  MoveC 4849 to (-301.47, 196.97, -44.5) mm, rotated rx -180 ry 0 rz 0.01 deg; joints [33.555, -39.251, 93.109, -140.852, 61.141, 159.518] to (-302.58, 195.21, -44.5) mm, rotated rx -180 ry 0 rz 0.01 deg; joints [33.481, -39.252, 93.114, -140.932, 61.116, 159.56]
  MoveL 4850 to (-302.58, 149.34, -44.5) mm, rotated rx -180 ry 0 rz 0.01 deg; joints [32.097, -40.399, 95.628, -142.863, 61.697, 161.24]
  MoveC 4851 to (-301.48, 145.02, -44.5) mm, rotated rx 180 ry 0 rz 0.01 deg; joints [31.985, -40.546, 95.95, -143.039, 61.798, 161.417] to (-298.46, 141.74, -44.5) mm, rotated rx 180 ry 0 rz 0.01 deg; joints [31.942, -40.745, 96.378, -143.159, 61.967, 161.595]
  MoveC 4852 to (-293.36, 138.32, -44.5) mm, rotated rx -180 ry 0 rz 0.01 deg; joints [31.935, -41.027, 96.986, -143.27, 62.225, 161.82] to (-288.34, 134.8, -44.5) mm, rotated rx 180 ry 0 rz 0.01 deg; joints [31.923, -41.306, 97.589, -143.384, 62.481, 162.044]
  MoveC 4853 to (-283.47, 131.07, -44.5) mm, rotated rx -180 ry 0 rz 0.01 deg; joints [31.901, -41.583, 98.188, -143.506, 62.732, 162.271] to (-278.83, 127.06, -44.5) mm, rotated rx -180 ry 0 rz 0.01 deg; joints [31.866, -41.856, 98.779, -143.64, 62.977, 162.5]
  MoveC 4854 to (-271.87, 120.15, -44.5) mm, rotated rx 180 ry 0 rz 0.01 deg; joints [31.785, -42.282, 99.704, -143.876, 63.353, 162.871] to (-265.5, 112.7, -44.5) mm, rotated rx -180 ry 0 rz 0.01 deg; joints [31.673, -42.694, 100.6, -144.136, 63.71, 163.243]
  MoveC 4855 to (-259.72, 104.78, -44.5) mm, rotated rx -180 ry 0 rz 0.01 deg; joints [31.534, -43.089, 101.465, -144.418, 64.048, 163.615] to (-254.52, 96.46, -44.5) mm, rotated rx 180 ry 0 rz 0.01 deg; joints [31.369, -43.468, 102.295, -144.719, 64.366, 163.983]
  MoveL 4856 to (-242.31, 74.19, -44.5) mm, rotated rx 180 ry 0 rz 0.01 deg; joints [30.883, -44.399, 104.348, -145.536, 65.145, 164.917]
  MoveC 4857 to (-239.21, 71.08, -44.5) mm, rotated rx 180 ry 0 rz 0.01 deg; joints [30.842, -44.578, 104.742, -145.635, 65.311, 165.069] to (-234.96, 69.94, -44.5) mm, rotated rx 180 ry 0 rz 0.01 deg; joints [30.888, -44.757, 105.133, -145.641, 65.498, 165.18]
  MoveL 4858 to (-158.58, 69.94, -44.5) mm, rotated rx 180 ry 0 rz 0.01 deg; joints [32.47, -47.442, 110.991, -144.753, 68.529, 166.484]
  MoveC 4859 to (-154.33, 71.08, -44.5) mm, rotated rx -180 ry 0 rz 0.01 deg; joints [32.601, -47.562, 111.253, -144.649, 68.678, 166.521] to (-151.22, 74.19, -44.5) mm, rotated rx -180 ry 0 rz 0.01 deg; joints [32.775, -47.603, 111.336, -144.479, 68.757, 166.48]
  MoveL 4860 to (-138.74, 96.86, -44.5) mm, rotated rx 180 ry 0 rz 0.01 deg; joints [33.818, -47.543, 111.16, -143.372, 68.936, 166.005]
  MoveC 4861 to (-132.58, 106.47, -44.5) mm, rotated rx -180 ry 0 rz 0.01 deg; joints [34.279, -47.541, 111.137, -142.891, 69.042, 165.816] to (-125.56, 115.48, -44.5) mm, rotated rx 180 ry 0 rz 0.01 deg; joints [34.74, -47.577, 111.197, -142.423, 69.186, 165.658]
  MoveC 4862 to (-117.83, 123.88, -44.5) mm, rotated rx -180 ry 0 rz 0.01 deg; joints [35.197, -47.646, 111.333, -141.967, 69.362, 165.53] to (-109.5, 131.68, -44.5) mm, rotated rx 180 ry 0 rz 0.01 deg; joints [35.65, -47.744, 111.532, -141.526, 69.566, 165.429]
  MoveC 4863 to (-106.07, 134.44, -44.5) mm, rotated rx 180 ry 0 rz 0.01 deg; joints [35.822, -47.793, 111.635, -141.362, 69.656, 165.402] to (-102.44, 136.93, -44.5) mm, rotated rx -180 ry 0 rz 0.01 deg; joints [35.99, -47.854, 111.765, -141.206, 69.756, 165.386]
  MoveC 4864 to (-98.74, 139.29, -44.5) mm, rotated rx 180 ry 0 rz 0.01 deg; joints [36.157, -47.92, 111.906, -141.053, 69.86, 165.375] to (-95.05, 141.69, -44.5) mm, rotated rx 180 ry 0 rz 0.01 deg; joints [36.324, -47.984, 112.042, -140.898, 69.962, 165.363]
  MoveC 4865 to (-92.03, 145, -44.5) mm, rotated rx -180 ry 0 rz 0.01 deg; joints [36.505, -48.006, 112.083, -140.717, 70.027, 165.311] to (-90.94, 149.34, -44.5) mm, rotated rx 180 ry 0 rz 0.01 deg; joints [36.673, -47.942, 111.934, -140.525, 70.008, 165.193]
  MoveL 4866 to (-90.94, 195.21, -44.5) mm, rotated rx 180 ry 0 rz 0.01 deg; joints [38.14, -46.86, 109.476, -138.699, 69.387, 163.706]
  MoveC 4867 to (-92.04, 196.97, -44.5) mm, rotated rx 180 ry 0 rz 0.01 deg; joints [38.168, -46.782, 109.301, -138.647, 69.323, 163.628] to (-94.11, 196.74, -44.5) mm, rotated rx -180 ry 0 rz 0.01 deg; joints [38.11, -46.721, 109.169, -138.688, 69.251, 163.599]
  MoveC 4868 to (-101.15, 191.39, -44.5) mm, rotated rx 180 ry 0 rz 0.01 deg; joints [37.77, -46.624, 108.966, -139.008, 69.068, 163.652] to (-108.38, 186.3, -44.5) mm, rotated rx 180 ry 0 rz 0.01 deg; joints [37.435, -46.512, 108.731, -139.319, 68.873, 163.692]
  MoveC 4869 to (-115.9, 181.63, -44.5) mm, rotated rx -180 ry 0 rz 0.01 deg; joints [37.108, -46.378, 108.447, -139.615, 68.66, 163.712] to (-123.75, 177.56, -44.5) mm, rotated rx 180 ry 0 rz 0.01 deg; joints [36.793, -46.216, 108.102, -139.891, 68.424, 163.706]
  MoveC 4870 to (-133.69, 173.48, -44.5) mm, rotated rx 180 ry 0 rz 0.01 deg; joints [36.431, -45.983, 107.602, -140.194, 68.109, 163.663] to (-143.98, 170.42, -44.5) mm, rotated rx -180 ry 0 rz 0.01 deg; joints [36.095, -45.71, 107.013, -140.457, 67.764, 163.578]
  MoveC 4871 to (-154.47, 168.17, -44.5) mm, rotated rx -180 ry 0 rz 0.01 deg; joints [35.784, -45.408, 106.36, -140.686, 67.398, 163.463] to (-165.06, 166.49, -44.5) mm, rotated rx -180 ry 0 rz 0.01 deg; joints [35.491, -45.084, 105.661, -140.888, 67.016, 163.325]
  MoveC 4872 to (-171.83, 165.83, -44.5) mm, rotated rx 180 ry 0 rz 0.01 deg; joints [35.319, -44.866, 105.189, -140.998, 66.766, 163.223] to (-178.62, 165.62, -44.5) mm, rotated rx 180 ry 0 rz 0.01 deg; joints [35.161, -44.635, 104.688, -141.088, 66.507, 163.106]
  MoveL 4873 to (-214.9, 165.62, -44.5) mm, rotated rx 180 ry 0 rz 0.01 deg; joints [34.374, -43.342, 101.899, -141.486, 65.088, 162.423]
  MoveC 4874 to (-230.33, 166.55, -44.5) mm, rotated rx 180 ry 0 rz 0.01 deg; joints [34.077, -42.755, 100.635, -141.597, 64.461, 162.093] to (-245.53, 169.34, -44.5) mm, rotated rx 180 ry 0 rz 0.01 deg; joints [33.847, -42.121, 99.271, -141.618, 63.812, 161.697]
  MoveL 4875 to (-245.78, 169.4, -44.5) mm, rotated rx 180 ry 0 rz 0.01 deg; joints [33.844, -42.11, 99.247, -141.618, 63.801, 161.69]
  MoveC 4876 to (-248.84, 171.23, -44.5) mm, rotated rx 180 ry 0 rz 0.01 deg; joints [33.837, -41.95, 98.902, -141.568, 63.653, 161.564] to (-250.35, 174.46, -44.5) mm, rotated rx 180 ry 0 rz 0.01 deg; joints [33.905, -41.814, 98.605, -141.447, 63.55, 161.42]
  MoveC 4877 to (-251.79, 177.71, -44.5) mm, rotated rx 180 ry 0 rz 0.01 deg; joints [33.974, -41.68, 98.312, -141.325, 63.45, 161.277] to (-254.71, 179.71, -44.5) mm, rotated rx 180 ry 0 rz 0.01 deg; joints [33.976, -41.519, 97.966, -141.265, 63.306, 161.146]
  MoveC 4878 to (-260.13, 181.68, -44.5) mm, rotated rx -180 ry 0 rz 0.01 deg; joints [33.925, -41.263, 97.416, -141.226, 63.059, 160.964] to (-265.46, 183.91, -44.5) mm, rotated rx 180 ry 0 rz 0.01 deg; joints [33.883, -41.003, 96.857, -141.174, 62.811, 160.774]
  MoveC 4879 to (-287.95, 196.94, -44.5) mm, rotated rx -180 ry 0 rz 0.01 deg; joints [33.822, -39.793, 94.259, -140.779, 61.711, 159.818] to (-307.16, 214.45, -44.5) mm, rotated rx -180 ry 0 rz 0.01 deg; joints [33.958, -38.561, 91.618, -140.142, 60.675, 158.723]
  MoveC 4880 to (-309.04, 214.92, -44.5) mm, rotated rx -180 ry 0 rz 0.01 deg; joints [33.934, -38.472, 91.428, -140.13, 60.589, 158.662] to (-310.14, 213.32, -44.5) mm, rotated rx 180 ry 0 rz 0.01 deg; joints [33.866, -38.469, 91.425, -140.203, 60.563, 158.698]
  MoveL 4881 to (-310.14, 144.76, -44.5) mm, rotated rx 180 ry 0 rz 0.01 deg; joints [31.812, -40.207, 95.227, -143.1, 61.432, 161.245]
  MoveC 4882 to (-309.04, 140.62, -44.5) mm, rotated rx 180 ry 0 rz 0.01 deg; joints [31.706, -40.35, 95.539, -143.268, 61.531, 161.416] to (-306.04, 137.56, -44.5) mm, rotated rx -180 ry 0 rz 0.01 deg; joints [31.668, -40.543, 95.955, -143.38, 61.697, 161.586]
  MoveC 4883 to (-295.24, 130.34, -44.5) mm, rotated rx 180 ry 0 rz 0.01 deg; joints [31.651, -41.141, 97.243, -143.617, 62.246, 162.06] to (-285.24, 122.05, -44.5) mm, rotated rx 180 ry 0 rz 0.01 deg; joints [31.585, -41.724, 98.504, -143.896, 62.771, 162.545]
  MoveC 4884 to (-276.09, 112.83, -44.5) mm, rotated rx 180 ry 0 rz 0.01 deg; joints [31.471, -42.287, 99.727, -144.215, 63.269, 163.036] to (-267.8, 102.84, -44.5) mm, rotated rx 180 ry 0 rz 0.01 deg; joints [31.314, -42.827, 100.905, -144.567, 63.738, 163.527]
  MoveC 4885 to (-264.28, 97.87, -44.5) mm, rotated rx -180 ry 0 rz 0.01 deg; joints [31.223, -43.07, 101.436, -144.745, 63.946, 163.757] to (-261.08, 92.69, -44.5) mm, rotated rx -180 ry 0 rz 0.01 deg; joints [31.119, -43.304, 101.95, -144.934, 64.143, 163.985]
  MoveL 4886 to (-246.68, 66.63, -44.5) mm, rotated rx 180 ry 0 rz 0.01 deg; joints [30.548, -44.397, 104.357, -145.893, 65.06, 165.077]
  MoveC 4887 to (-243.58, 63.52, -44.5) mm, rotated rx -180 ry 0 rz 0.01 deg; joints [30.506, -44.576, 104.751, -145.993, 65.226, 165.229] to (-239.33, 62.38, -44.5) mm, rotated rx -180 ry 0 rz 0.01 deg; joints [30.551, -44.755, 105.142, -146, 65.414, 165.338]
  MoveL 4888 to (-154.21, 62.38, -44.5) mm, rotated rx -180 ry 0 rz 0.01 deg; joints [32.307, -47.744, 111.671, -145.008, 68.796, 166.781]
  MoveC 4889 to (-149.96, 63.52, -44.5) mm, rotated rx -180 ry 0 rz 0.01 deg; joints [32.438, -47.864, 111.932, -144.903, 68.945, 166.817] to (-146.85, 66.63, -44.5) mm, rotated rx -180 ry 0 rz 0.01 deg; joints [32.613, -47.904, 112.016, -144.732, 69.024, 166.777]
  MoveL 4890 to (-132.19, 93.08, -44.5) mm, rotated rx 180 ry 0 rz 0.01 deg; joints [33.839, -47.841, 111.823, -143.435, 69.234, 166.23]
  MoveC 4891 to (-123.29, 106.29, -44.5) mm, rotated rx 180 ry 0 rz 0.01 deg; joints [34.486, -47.852, 111.819, -142.764, 69.393, 165.979] to (-112.66, 118.15, -44.5) mm, rotated rx 180 ry 0 rz 0.01 deg; joints [35.128, -47.941, 111.992, -142.122, 69.631, 165.795]
  MoveC 4892 to (-100.62, 128.57, -44.5) mm, rotated rx -180 ry 0 rz 0.01 deg; joints [35.758, -48.1, 112.322, -141.515, 69.936, 165.678] to (-87.47, 137.53, -44.5) mm, rotated rx -180 ry 0 rz 0.01 deg; joints [36.371, -48.319, 112.79, -140.944, 70.295, 165.623]
  MoveC 4893 to (-84.47, 140.62, -44.5) mm, rotated rx 180 ry 0 rz 0.01 deg; joints [36.545, -48.345, 112.841, -140.772, 70.362, 165.578] to (-83.38, 144.77, -44.5) mm, rotated rx 180 ry 0 rz 0.01 deg; joints [36.708, -48.286, 112.701, -140.587, 70.345, 165.466]
  MoveL 4894 to (-83.38, 213.32, -44.5) mm, rotated rx 180 ry 0 rz 0.01 deg; joints [38.891, -46.656, 108.998, -137.867, 69.413, 163.235]
  MoveC 4895 to (-84.48, 214.91, -44.5) mm, rotated rx -180 ry 0 rz 0.01 deg; joints [38.913, -46.582, 108.832, -137.822, 69.352, 163.161] to (-86.36, 214.45, -44.5) mm, rotated rx 180 ry 0 rz 0.01 deg; joints [38.852, -46.533, 108.727, -137.87, 69.291, 163.143]
  MoveC 4896 to (-103.09, 198.94, -44.5) mm, rotated rx 180 ry 0 rz 0.01 deg; joints [37.959, -46.377, 108.414, -138.738, 68.896, 163.365] to (-122.53, 187, -44.5) mm, rotated rx -180 ry 0 rz 0.01 deg; joints [37.119, -46.03, 107.679, -139.497, 68.343, 163.415]
  MoveC 4897 to (-143.76, 178.74, -44.5) mm, rotated rx -180 ry 0 rz 0.01 deg; joints [36.363, -45.519, 106.583, -140.12, 67.662, 163.306] to (-166.04, 173.99, -44.5) mm, rotated rx 180 ry 0 rz 0.01 deg; joints [35.705, -44.872, 105.187, -140.597, 66.881, 163.057]
  MoveC 4898 to (-172.31, 173.38, -44.5) mm, rotated rx 180 ry 0 rz 0.01 deg; joints [35.545, -44.669, 104.749, -140.698, 66.648, 162.962] to (-178.62, 173.18, -44.5) mm, rotated rx 180 ry 0 rz 0.01 deg; joints [35.398, -44.454, 104.284, -140.781, 66.409, 162.851]
  MoveL 4899 to (-214.9, 173.18, -44.5) mm, rotated rx 180 ry 0 rz 0.01 deg; joints [34.608, -43.16, 101.494, -141.176, 64.991, 162.164]
  MoveC 4900 to (-235.07, 174.82, -44.5) mm, rotated rx -180 ry 0 rz 0.01 deg; joints [34.233, -42.378, 99.812, -141.301, 64.164, 161.713] to (-254.71, 179.71, -44.5) mm, rotated rx 180 ry 0 rz 0.01 deg; joints [33.976, -41.519, 97.966, -141.265, 63.306, 161.146]
  MoveC 4901 to (-257.49, 181.72, -44.5) mm, rotated rx 180 ry 0 rz 0.01 deg; joints [33.979, -41.363, 97.63, -141.204, 63.166, 161.017] to (-258.67, 184.93, -44.5) mm, rotated rx -180 ry 0 rz 0.01 deg; joints [34.053, -41.238, 97.357, -141.08, 63.077, 160.878]
  MoveC 4902 to (-259.76, 188.16, -44.5) mm, rotated rx -180 ry 0 rz 0.01 deg; joints [34.128, -41.115, 97.089, -140.955, 62.991, 160.739] to (-262.38, 190.33, -44.5) mm, rotated rx -180 ry 0 rz 0.01 deg; joints [34.14, -40.96, 96.754, -140.884, 62.856, 160.606]
  MoveC 4903 to (-291.82, 209.03, -44.5) mm, rotated rx 180 ry 0 rz 0.01 deg; joints [34.103, -39.324, 93.244, -140.294, 61.394, 159.279] to (-314.46, 235.55, -44.5) mm, rotated rx -180 ry 0 rz 0.01 deg; joints [34.426, -37.687, 89.738, -139.276, 60.092, 157.725]
  MoveC 4904 to (-316.16, 236.21, -44.5) mm, rotated rx -180 ry 0 rz 0.01 deg; joints [34.412, -37.599, 89.55, -139.254, 60.011, 157.658] to (-317.25, 234.75, -44.5) mm, rotated rx 180 ry 0 rz 0.01 deg; joints [34.348, -37.593, 89.54, -139.32, 59.982, 157.689]
  MoveL 4905 to (-317.25, 140.22, -44.5) mm, rotated rx -180 ry 0 rz 0.01 deg; joints [31.538, -40.029, 94.857, -143.33, 61.184, 161.257]
  MoveC 4906 to (-316.15, 136.26, -44.5) mm, rotated rx -180 ry 0 rz 0.01 deg; joints [31.437, -40.168, 95.159, -143.491, 61.28, 161.422] to (-313.18, 133.42, -44.5) mm, rotated rx 180 ry 0 rz 0.01 deg; joints [31.406, -40.355, 95.562, -143.595, 61.443, 161.584]
  MoveC 4907 to (-301.85, 126.44, -44.5) mm, rotated rx -180 ry 0 rz 0.01 deg; joints [31.404, -40.971, 96.887, -143.823, 62.014, 162.062] to (-291.44, 118.13, -44.5) mm, rotated rx -180 ry 0 rz 0.01 deg; joints [31.342, -41.572, 98.186, -144.104, 62.558, 162.557]
  MoveC 4908 to (-281.99, 108.76, -44.5) mm, rotated rx 180 ry 0 rz 0.01 deg; joints [31.228, -42.152, 99.444, -144.429, 63.072, 163.059] to (-273.47, 98.55, -44.5) mm, rotated rx 180 ry 0 rz 0.01 deg; joints [31.066, -42.706, 100.653, -144.792, 63.556, 163.562]
  MoveC 4909 to (-270.21, 93.94, -44.5) mm, rotated rx -180 ry 0 rz 0.01 deg; joints [30.982, -42.932, 101.146, -144.958, 63.749, 163.775] to (-267.24, 89.14, -44.5) mm, rotated rx -180 ry 0 rz 0.01 deg; joints [30.884, -43.149, 101.622, -145.134, 63.932, 163.987]
  MoveL 4910 to (-250.77, 59.48, -44.5) mm, rotated rx 180 ry 0 rz 0.01 deg; joints [30.232, -44.394, 104.364, -146.23, 64.981, 165.228]
  MoveC 4911 to (-247.69, 56.39, -44.5) mm, rotated rx 180 ry 0 rz 0.01 deg; joints [30.189, -44.571, 104.754, -146.33, 65.146, 165.378] to (-243.48, 55.27, -44.5) mm, rotated rx 180 ry 0 rz 0.01 deg; joints [30.233, -44.749, 105.143, -146.338, 65.333, 165.486]
  MoveL 4912 to (-150.04, 55.27, -44.5) mm, rotated rx 180 ry 0 rz 0.01 deg; joints [32.152, -48.028, 112.311, -145.247, 69.05, 167.058]
  MoveC 4913 to (-145.85, 56.39, -44.5) mm, rotated rx 180 ry 0 rz 0.01 deg; joints [32.282, -48.145, 112.568, -145.142, 69.197, 167.094] to (-142.78, 59.46, -44.5) mm, rotated rx -180 ry 0 rz 0.01 deg; joints [32.455, -48.186, 112.652, -144.972, 69.275, 167.055]
  MoveL 4914 to (-126.04, 89.52, -44.5) mm, rotated rx 180 ry 0 rz 0.01 deg; joints [33.858, -48.119, 112.443, -143.491, 69.514, 166.441]
  MoveC 4915 to (-117.03, 102.79, -44.5) mm, rotated rx -180 ry 0 rz 0.01 deg; joints [34.513, -48.131, 112.443, -142.814, 69.675, 166.191] to (-106.22, 114.63, -44.5) mm, rotated rx -180 ry 0 rz 0.01 deg; joints [35.162, -48.226, 112.628, -142.167, 69.917, 166.012]
  MoveC 4916 to (-93.89, 124.88, -44.5) mm, rotated rx 180 ry 0 rz 0.01 deg; joints [35.796, -48.397, 112.985, -141.558, 70.233, 165.906] to (-80.33, 133.42, -44.5) mm, rotated rx 180 ry 0 rz 0.01 deg; joints [36.409, -48.637, 113.5, -140.993, 70.61, 165.872]
  MoveC 4917 to (-77.36, 136.28, -44.5) mm, rotated rx 180 ry 0 rz 0.01 deg; joints [36.576, -48.667, 113.56, -140.829, 70.679, 165.834] to (-76.26, 140.26, -44.5) mm, rotated rx -180 ry 0 rz 0.01 deg; joints [36.734, -48.612, 113.431, -140.651, 70.664, 165.728]
  MoveL 4918 to (-76.26, 234.75, -44.5) mm, rotated rx -180 ry 0 rz 0.01 deg; joints [39.726, -46.342, 108.276, -136.917, 69.377, 162.633]
  MoveC 4919 to (-77.36, 236.2, -44.5) mm, rotated rx -180 ry 0 rz 0.01 deg; joints [39.743, -46.27, 108.116, -136.878, 69.318, 162.563] to (-79.06, 235.54, -44.5) mm, rotated rx 180 ry 0 rz 0.01 deg; joints [39.68, -46.233, 108.036, -136.93, 69.267, 162.555]
  MoveC 4920 to (-91.63, 218.9, -44.5) mm, rotated rx -180 ry 0 rz 0.01 deg; joints [38.858, -46.253, 108.107, -137.777, 69.042, 162.897] to (-107.02, 204.82, -44.5) mm, rotated rx 180 ry 0 rz 0.01 deg; joints [38.047, -46.104, 107.809, -138.563, 68.674, 163.097]
  MoveC 4921 to (-124.62, 193.66, -44.5) mm, rotated rx -180 ry 0 rz 0.01 deg; joints [37.278, -45.799, 107.164, -139.261, 68.177, 163.154] to (-143.84, 185.59, -44.5) mm, rotated rx 180 ry 0 rz 0.01 deg; joints [36.575, -45.351, 106.206, -139.846, 67.569, 163.075]
  MoveC 4922 to (-161.28, 181.45, -44.5) mm, rotated rx 180 ry 0 rz 0.01 deg; joints [36.046, -44.856, 105.14, -140.237, 66.964, 162.894] to (-179.16, 180.15, -44.5) mm, rotated rx -180 ry 0 rz 0.01 deg; joints [35.604, -44.267, 103.867, -140.505, 66.297, 162.605]
  MoveL 4923 to (-214.9, 180.29, -44.5) mm, rotated rx 180 ry 0 rz 0.01 deg; joints [34.828, -42.986, 101.109, -140.885, 64.899, 161.918]
  MoveC 4924 to (-239.16, 182.83, -44.5) mm, rotated rx -180 ry 0 rz 0.01 deg; joints [34.392, -42.028, 99.05, -141.008, 63.897, 161.35] to (-262.38, 190.33, -44.5) mm, rotated rx -180 ry 0 rz 0.01 deg; joints [34.14, -40.96, 96.754, -140.884, 62.856, 160.606]
  MoveC 4925 to (-264.75, 192.39, -44.5) mm, rotated rx -180 ry 0 rz 0.01 deg; joints [34.154, -40.817, 96.445, -140.816, 62.732, 160.482] to (-265.56, 195.42, -44.5) mm, rotated rx -180 ry 0 rz 0.01 deg; joints [34.228, -40.708, 96.209, -140.696, 62.66, 160.354]
  MoveC 4926 to (-266.3, 198.45, -44.5) mm, rotated rx 180 ry 0 rz 0.01 deg; joints [34.304, -40.602, 95.979, -140.576, 62.591, 160.228] to (-268.52, 200.64, -44.5) mm, rotated rx 180 ry 0 rz 0.01 deg; joints [34.324, -40.46, 95.672, -140.5, 62.471, 160.1]
  MoveC 4927 to (-298.38, 224.61, -44.5) mm, rotated rx -180 ry 0 rz 0.01 deg; joints [34.429, -38.645, 91.78, -139.672, 60.917, 158.533] to (-318.34, 257.3, -44.5) mm, rotated rx -180 ry 0 rz 0.01 deg; joints [34.971, -36.913, 88.072, -138.361, 59.643, 156.751]
  MoveC 4928 to (-321.51, 259.04, -44.5) mm, rotated rx 180 ry 0 rz 0.01 deg; joints [34.957, -36.73, 87.682, -138.295, 59.484, 156.6] to (-323.82, 256.26, -44.5) mm, rotated rx -180 ry 0 rz 0.01 deg; joints [34.833, -36.712, 87.649, -138.42, 59.42, 156.656]
  MoveL 4929 to (-323.82, 135.82, -44.5) mm, rotated rx 180 ry 0 rz 0.01 deg; joints [31.28, -39.868, 94.522, -143.549, 60.955, 161.276]
  MoveC 4930 to (-322.72, 132.02, -44.5) mm, rotated rx 180 ry 0 rz 0.01 deg; joints [31.184, -40.003, 94.816, -143.705, 61.05, 161.434] to (-319.76, 129.4, -44.5) mm, rotated rx -180 ry 0 rz 0.01 deg; joints [31.158, -40.185, 95.207, -143.801, 61.21, 161.589]
  MoveC 4931 to (-307.94, 122.71, -44.5) mm, rotated rx 180 ry 0 rz 0.01 deg; joints [31.172, -40.816, 96.563, -144.017, 61.801, 162.068] to (-297.15, 114.45, -44.5) mm, rotated rx 180 ry 0 rz 0.01 deg; joints [31.118, -41.433, 97.895, -144.297, 62.363, 162.569]
  MoveC 4932 to (-287.43, 104.98, -44.5) mm, rotated rx -180 ry 0 rz 0.01 deg; joints [31.004, -42.026, 99.182, -144.628, 62.891, 163.081] to (-278.71, 94.58, -44.5) mm, rotated rx 180 ry 0 rz 0.01 deg; joints [30.839, -42.593, 100.417, -144.999, 63.386, 163.594]
  MoveC 4933 to (-275.68, 90.31, -44.5) mm, rotated rx -180 ry 0 rz 0.01 deg; joints [30.76, -42.803, 100.875, -145.154, 63.565, 163.791] to (-272.93, 85.86, -44.5) mm, rotated rx 180 ry 0 rz 0.01 deg; joints [30.669, -43.004, 101.317, -145.318, 63.736, 163.988]
  MoveL 4934 to (-254.5, 52.76, -44.5) mm, rotated rx 180 ry 0 rz 0.01 deg; joints [29.937, -44.394, 104.377, -146.546, 64.91, 165.371]
  MoveC 4935 to (-251.61, 49.79, -44.5) mm, rotated rx 180 ry 0 rz 0.01 deg; joints [29.894, -44.561, 104.746, -146.644, 65.066, 165.514] to (-247.62, 48.7, -44.5) mm, rotated rx 180 ry 0 rz 0.01 deg; joints [29.934, -44.731, 105.116, -146.652, 65.244, 165.617]
  MoveL 4936 to (-145.87, 48.7, -44.5) mm, rotated rx -180 ry 0 rz 0.01 deg; joints [32.015, -48.298, 112.922, -145.463, 69.297, 167.318]
  MoveC 4937 to (-141.9, 49.79, -44.5) mm, rotated rx -180 ry 0 rz 0.01 deg; joints [32.14, -48.409, 113.165, -145.362, 69.436, 167.351] to (-139.04, 52.76, -44.5) mm, rotated rx 180 ry 0 rz 0.01 deg; joints [32.306, -48.445, 113.238, -145.198, 69.507, 167.311]
  MoveL 4938 to (-120.09, 86.14, -44.5) mm, rotated rx 180 ry 0 rz 0.01 deg; joints [33.879, -48.385, 113.036, -143.542, 69.783, 166.641]
  MoveC 4939 to (-109.01, 101.89, -44.5) mm, rotated rx -180 ry 0 rz 0.01 deg; joints [34.669, -48.411, 113.063, -142.729, 69.986, 166.353] to (-95.55, 115.66, -44.5) mm, rotated rx -180 ry 0 rz 0.01 deg; joints [35.449, -48.546, 113.334, -141.958, 70.297, 166.161]
  MoveC 4940 to (-90.49, 119.69, -44.5) mm, rotated rx 180 ry 0 rz 0.01 deg; joints [35.705, -48.619, 113.488, -141.714, 70.428, 166.123] to (-85.1, 123.27, -44.5) mm, rotated rx 180 ry 0 rz 0.01 deg; joints [35.955, -48.712, 113.685, -141.481, 70.576, 166.104]
  MoveC 4941 to (-79.49, 126.48, -44.5) mm, rotated rx -180 ry 0 rz 0.01 deg; joints [36.198, -48.818, 113.914, -141.259, 70.736, 166.1] to (-73.74, 129.42, -44.5) mm, rotated rx 180 ry 0 rz 0.01 deg; joints [36.437, -48.933, 114.164, -141.044, 70.903, 166.106]
  MoveC 4942 to (-70.79, 132.06, -44.5) mm, rotated rx -180 ry 0 rz 0.01 deg; joints [36.598, -48.967, 114.233, -140.888, 70.973, 166.075] to (-69.69, 135.86, -44.5) mm, rotated rx -180 ry 0 rz 0.01 deg; joints [36.751, -48.916, 114.113, -140.717, 70.96, 165.976]
  MoveL 4943 to (-69.7, 256.24, -44.5) mm, rotated rx 180 ry 0 rz 0.01 deg; joints [40.54, -45.994, 107.48, -135.979, 69.319, 162.005]
  MoveC 4944 to (-72.01, 259.03, -44.5) mm, rotated rx -180 ry 0 rz 0.01 deg; joints [40.564, -45.848, 107.157, -135.908, 69.2, 161.865] to (-75.18, 257.28, -44.5) mm, rotated rx -180 ry 0 rz 0.01 deg; joints [40.432, -45.793, 107.041, -136.025, 69.111, 161.868]
  MoveC 4945 to (-84.92, 238.26, -44.5) mm, rotated rx -180 ry 0 rz 0.01 deg; joints [39.615, -45.976, 107.472, -136.916, 69.021, 162.354] to (-98.2, 221.52, -44.5) mm, rotated rx 180 ry 0 rz 0.01 deg; joints [38.776, -45.974, 107.497, -137.774, 68.77, 162.689]
  MoveC 4946 to (-114.38, 207.58, -44.5) mm, rotated rx 180 ry 0 rz 0.01 deg; joints [37.954, -45.795, 107.13, -138.562, 68.368, 162.87] to (-132.8, 196.78, -44.5) mm, rotated rx 180 ry 0 rz 0.01 deg; joints [37.181, -45.45, 106.4, -139.25, 67.833, 162.9]
  MoveC 4947 to (-152.55, 189.9, -44.5) mm, rotated rx -180 ry 0 rz 0.01 deg; joints [36.508, -44.95, 105.329, -139.787, 67.184, 162.769] to (-173.3, 187.29, -44.5) mm, rotated rx 180 ry 0 rz 0.01 deg; joints [35.956, -44.298, 103.922, -140.148, 66.429, 162.472]
  MoveL 4948 to (-214.9, 186.86, -44.5) mm, rotated rx -180 ry 0 rz 0.01 deg; joints [35.03, -42.825, 100.75, -140.617, 64.814, 161.689]
  MoveC 4949 to (-242.58, 190.36, -44.5) mm, rotated rx -180 ry 0 rz 0.01 deg; joints [34.55, -41.712, 98.361, -140.727, 63.662, 161.013] to (-268.52, 200.64, -44.5) mm, rotated rx 180 ry 0 rz 0.01 deg; joints [34.324, -40.46, 95.672, -140.5, 62.471, 160.1]
  MoveC 4950 to (-271.62, 203.85, -44.5) mm, rotated rx -180 ry 0 rz 0.01 deg; joints [34.357, -40.257, 95.234, -140.388, 62.302, 159.915] to (-272.38, 208.25, -44.5) mm, rotated rx -180 ry 0 rz 0.01 deg; joints [34.472, -40.113, 94.921, -140.21, 62.214, 159.735]
  MoveC 4951 to (-272.98, 212.62, -44.5) mm, rotated rx 180 ry 0 rz 0.01 deg; joints [34.589, -39.975, 94.621, -140.032, 62.133, 159.559] to (-275.74, 216.08, -44.5) mm, rotated rx 180 ry 0 rz 0.01 deg; joints [34.635, -39.776, 94.193, -139.905, 61.975, 159.369]
  MoveC 4952 to (-297.18, 237.6, -44.5) mm, rotated rx 180 ry 0 rz 0.01 deg; joints [34.829, -38.34, 91.114, -139.119, 60.8, 158.054] to (-311.04, 264.63, -44.5) mm, rotated rx -180 ry 0 rz 0.01 deg; joints [35.324, -37.008, 88.261, -138.026, 59.861, 156.633]
  MoveC 4953 to (-313.15, 267.5, -44.5) mm, rotated rx 180 ry 0 rz 0.01 deg; joints [35.362, -36.837, 87.896, -137.91, 59.733, 156.462] to (-316.53, 268.6, -44.5) mm, rotated rx 180 ry 0 rz 0.01 deg; joints [35.326, -36.663, 87.527, -137.872, 59.573, 156.331]
  MoveL 4954 to (-329.33, 268.6, -44.5) mm, rotated rx 180 ry 0 rz 0.01 deg; joints [35.072, -36.119, 86.383, -137.9, 59.02, 156.002]
  MoveC 4955 to (-332.06, 267.47, -44.5) mm, rotated rx -180 ry 0 rz 0.01 deg; joints [34.987, -36.036, 86.209, -137.953, 58.916, 155.978] to (-333.18, 264.75, -44.5) mm, rotated rx -180 ry 0 rz 0.01 deg; joints [34.888, -36.067, 86.278, -138.073, 58.902, 156.063]
  MoveL 4956 to (-333.18, 129.66, -44.5) mm, rotated rx 180 ry 0 rz 0.01 deg; joints [30.918, -39.632, 94.031, -143.855, 60.625, 161.297]
  MoveC 4957 to (-332.04, 125.85, -44.5) mm, rotated rx 180 ry 0 rz 0.01 deg; joints [30.821, -39.769, 94.328, -144.012, 60.722, 161.457] to (-329.01, 123.27, -44.5) mm, rotated rx 180 ry 0 rz 0.01 deg; joints [30.798, -39.954, 94.726, -144.107, 60.886, 161.613]
  MoveC 4958 to (-324.12, 121.05, -44.5) mm, rotated rx 180 ry 0 rz 0.01 deg; joints [30.819, -40.205, 95.263, -144.177, 61.125, 161.793] to (-319.29, 118.71, -44.5) mm, rotated rx 180 ry 0 rz 0.01 deg; joints [30.836, -40.454, 95.799, -144.251, 61.363, 161.975]
  MoveC 4959 to (-314.57, 116.14, -44.5) mm, rotated rx -180 ry 0 rz 0.01 deg; joints [30.843, -40.703, 96.334, -144.333, 61.598, 162.161] to (-310.05, 113.24, -44.5) mm, rotated rx -180 ry 0 rz 0.01 deg; joints [30.837, -40.95, 96.866, -144.429, 61.828, 162.353]
  MoveC 4960 to (-294.8, 99.95, -44.5) mm, rotated rx -180 ry 0 rz 0.01 deg; joints [30.704, -41.852, 98.817, -144.891, 62.642, 163.107] to (-282.84, 83.64, -44.5) mm, rotated rx 180 ry 0 rz 0.01 deg; joints [30.409, -42.674, 100.61, -145.489, 63.348, 163.876]
  MoveL 4961 to (-263.19, 49.54, -44.5) mm, rotated rx 180 ry 0 rz 0.01 deg; joints [29.665, -44.135, 103.825, -146.759, 64.589, 165.319]
  MoveC 4962 to (-262.37, 48.03, -44.5) mm, rotated rx 180 ry 0 rz 0.01 deg; joints [29.63, -44.196, 103.96, -146.815, 64.641, 165.38] to (-261.64, 46.49, -44.5) mm, rotated rx -180 ry 0 rz 0.01 deg; joints [29.593, -44.255, 104.09, -146.874, 64.691, 165.441]
  MoveC 4963 to (-260.95, 44.92, -44.5) mm, rotated rx 180 ry 0 rz 0.01 deg; joints [29.554, -44.313, 104.218, -146.933, 64.739, 165.501] to (-260.24, 43.36, -44.5) mm, rotated rx 180 ry 0 rz 0.01 deg; joints [29.515, -44.371, 104.346, -146.993, 64.787, 165.562]
  MoveC 4964 to (-257.69, 40.43, -44.5) mm, rotated rx -180 ry 0 rz 0.01 deg; joints [29.465, -44.525, 104.686, -147.093, 64.929, 165.696] to (-253.96, 39.33, -44.5) mm, rotated rx 180 ry 0 rz 0.01 deg; joints [29.499, -44.685, 105.035, -147.105, 65.097, 165.794]
  MoveL 4965 to (-139.53, 39.33, -44.5) mm, rotated rx 180 ry 0 rz 0.01 deg; joints [31.826, -48.694, 113.818, -145.764, 69.664, 167.69]
  MoveC 4966 to (-135.8, 40.43, -44.5) mm, rotated rx -180 ry 0 rz 0.01 deg; joints [31.946, -48.796, 114.041, -145.665, 69.793, 167.718] to (-133.26, 43.38, -44.5) mm, rotated rx 180 ry 0 rz 0.01 deg; joints [32.105, -48.822, 114.093, -145.506, 69.852, 167.675]
  MoveC 4967 to (-132.51, 45.05, -44.5) mm, rotated rx 180 ry 0 rz 0.01 deg; joints [32.18, -48.813, 114.071, -145.425, 69.858, 167.639] to (-131.77, 46.72, -44.5) mm, rotated rx 180 ry 0 rz 0.01 deg; joints [32.255, -48.805, 114.048, -145.345, 69.864, 167.603]
  MoveC 4968 to (-130.99, 48.38, -44.5) mm, rotated rx -180 ry 0 rz 0.01 deg; joints [32.331, -48.798, 114.029, -145.264, 69.872, 167.568] to (-130.12, 49.99, -44.5) mm, rotated rx -180 ry 0 rz 0.01 deg; joints [32.406, -48.794, 114.018, -145.185, 69.884, 167.536]
  MoveL 4969 to (-109.64, 85.01, -44.5) mm, rotated rx 180 ry 0 rz 0.01 deg; joints [34.081, -48.748, 113.842, -143.43, 70.189, 166.848]
  MoveC 4970 to (-97.35, 101.31, -44.5) mm, rotated rx 180 ry 0 rz 0.01 deg; joints [34.923, -48.798, 113.921, -142.571, 70.426, 166.565] to (-81.73, 114.45, -44.5) mm, rotated rx 180 ry 0 rz 0.01 deg; joints [35.741, -49.011, 114.366, -141.783, 70.819, 166.429]
  MoveC 4971 to (-77.6, 117, -44.5) mm, rotated rx 180 ry 0 rz 0.01 deg; joints [35.927, -49.085, 114.525, -141.611, 70.934, 166.421] to (-73.32, 119.26, -44.5) mm, rotated rx -180 ry 0 rz 0.01 deg; joints [36.108, -49.17, 114.709, -141.448, 71.058, 166.424]
  MoveC 4972 to (-68.93, 121.33, -44.5) mm, rotated rx -180 ry 0 rz 0.01 deg; joints [36.285, -49.262, 114.908, -141.29, 71.188, 166.435] to (-64.5, 123.28, -44.5) mm, rotated rx 180 ry 0 rz 0.01 deg; joints [36.46, -49.357, 115.116, -141.135, 71.321, 166.45]
  MoveC 4973 to (-61.47, 125.8, -44.5) mm, rotated rx 180 ry 0 rz 0.01 deg; joints [36.62, -49.395, 115.196, -140.981, 71.395, 166.424] to (-60.33, 129.57, -44.5) mm, rotated rx 180 ry 0 rz 0.01 deg; joints [36.775, -49.347, 115.081, -140.809, 71.383, 166.327]
  MoveL 4974 to (-60.33, 264.75, -44.5) mm, rotated rx 180 ry 0 rz 0.01 deg; joints [41.034, -46.064, 107.619, -135.5, 69.532, 161.876]
  MoveC 4975 to (-61.46, 267.48, -44.5) mm, rotated rx 180 ry 0 rz 0.01 deg; joints [41.085, -45.957, 107.381, -135.414, 69.456, 161.759] to (-64.19, 268.61, -44.5) mm, rotated rx -180 ry 0 rz 0.01 deg; joints [41.048, -45.841, 107.127, -135.414, 69.345, 161.669]
  MoveL 4976 to (-76.98, 268.61, -44.5) mm, rotated rx -180 ry 0 rz 0.01 deg; joints [40.722, -45.435, 106.247, -135.616, 68.896, 161.434]
  MoveC 4977 to (-80.37, 267.51, -44.5) mm, rotated rx 180 ry 0 rz 0.01 deg; joints [40.604, -45.356, 106.077, -135.711, 68.79, 161.41] to (-82.47, 264.64, -44.5) mm, rotated rx 180 ry 0 rz 0.01 deg; joints [40.466, -45.365, 106.101, -135.854, 68.754, 161.473]
  MoveC 4978 to (-91.05, 245.84, -44.5) mm, rotated rx -180 ry 0 rz 0.01 deg; joints [39.69, -45.583, 106.605, -136.714, 68.7, 161.978] to (-103.51, 229.35, -44.5) mm, rotated rx 180 ry 0 rz 0.01 deg; joints [38.885, -45.603, 106.676, -137.545, 68.473, 162.323]
  MoveC 4979 to (-119.02, 215.74, -44.5) mm, rotated rx -180 ry 0 rz 0.01 deg; joints [38.094, -45.438, 106.341, -138.305, 68.089, 162.506] to (-136.79, 205.25, -44.5) mm, rotated rx -180 ry 0 rz 0.01 deg; joints [37.349, -45.107, 105.641, -138.966, 67.572, 162.538]
  MoveC 4980 to (-155.59, 198.76, -44.5) mm, rotated rx 180 ry 0 rz 0.01 deg; joints [36.713, -44.629, 104.617, -139.47, 66.952, 162.411] to (-175.34, 196.42, -44.5) mm, rotated rx 180 ry 0 rz 0.01 deg; joints [36.192, -44.002, 103.266, -139.803, 66.231, 162.119]
  MoveL 4981 to (-214.9, 196.22, -44.5) mm, rotated rx 180 ry 0 rz 0.01 deg; joints [35.315, -42.592, 100.234, -140.235, 64.693, 161.36]
  MoveC 4982 to (-245.9, 200.99, -44.5) mm, rotated rx 180 ry 0 rz 0.01 deg; joints [34.802, -41.318, 97.501, -140.316, 63.391, 160.562] to (-274.04, 214.87, -44.5) mm, rotated rx 180 ry 0 rz 0.01 deg; joints [34.634, -39.875, 94.404, -139.945, 62.061, 159.452]
  MoveC 4983 to (-274.89, 215.47, -44.5) mm, rotated rx 180 ry 0 rz 0.01 deg; joints [34.635, -39.826, 94.298, -139.925, 62.018, 159.41] to (-275.74, 216.08, -44.5) mm, rotated rx -180 ry 0 rz 0.01 deg; joints [34.635, -39.776, 94.193, -139.905, 61.975, 159.369]
  MoveC 4984 to (-278.58, 219.93, -44.5) mm, rotated rx 180 ry 0 rz 0.01 deg; joints [34.691, -39.562, 93.732, -139.762, 61.807, 159.16] to (-278.72, 224.71, -44.5) mm, rotated rx 180 ry 0 rz 0.01 deg; joints [34.828, -39.429, 93.442, -139.563, 61.74, 158.975]
  MoveC 4985 to (-278.68, 229.44, -44.5) mm, rotated rx 180 ry 0 rz 0.01 deg; joints [34.967, -39.304, 93.169, -139.365, 61.68, 158.795] to (-281.02, 233.55, -44.5) mm, rotated rx 180 ry 0 rz 0.01 deg; joints [35.039, -39.1, 92.73, -139.207, 61.53, 158.584]
  MoveC 4986 to (-283.38, 236.01, -44.5) mm, rotated rx -180 ry 0 rz 0.01 deg; joints [35.063, -38.939, 92.385, -139.117, 61.4, 158.435] to (-285.66, 238.55, -44.5) mm, rotated rx 180 ry 0 rz 0.01 deg; joints [35.09, -38.779, 92.041, -139.023, 61.272, 158.284]
  MoveC 4987 to (-296.89, 255.15, -44.5) mm, rotated rx 180 ry 0 rz 0.01 deg; joints [35.339, -37.863, 90.079, -138.377, 60.585, 157.364] to (-303.91, 273.92, -44.5) mm, rotated rx 180 ry 0 rz 0.01 deg; joints [35.729, -37.036, 88.305, -137.608, 60.043, 156.429]
  MoveC 4988 to (-305.79, 276.83, -44.5) mm, rotated rx -180 ry 0 rz 0.01 deg; joints [35.772, -36.873, 87.957, -137.49, 59.925, 156.261] to (-309.06, 277.96, -44.5) mm, rotated rx -180 ry 0 rz 0.01 deg; joints [35.738, -36.703, 87.598, -137.452, 59.771, 156.132]
  MoveL 4989 to (-338.69, 277.96, -44.5) mm, rotated rx 180 ry 0 rz 0.01 deg; joints [35.15, -35.437, 84.936, -137.506, 58.488, 155.356]
  MoveC 4990 to (-341.42, 276.83, -44.5) mm, rotated rx -180 ry 0 rz 0.01 deg; joints [35.065, -35.352, 84.759, -137.557, 58.383, 155.331] to (-342.55, 274.11, -44.5) mm, rotated rx 180 ry 0 rz 0.01 deg; joints [34.967, -35.384, 84.831, -137.677, 58.369, 155.417]
  MoveL 4991 to (-342.54, 123.02, -44.5) mm, rotated rx 180 ry 0 rz 0.01 deg; joints [30.542, -39.403, 93.556, -144.178, 60.297, 161.334]
  MoveC 4992 to (-341.45, 119.49, -44.5) mm, rotated rx 180 ry 0 rz 0.01 deg; joints [30.453, -39.531, 93.834, -144.324, 60.388, 161.484] to (-338.57, 117.19, -44.5) mm, rotated rx 180 ry 0 rz 0.01 deg; joints [30.435, -39.704, 94.206, -144.41, 60.544, 161.627]
  MoveC 4993 to (-332.56, 114.71, -44.5) mm, rotated rx 180 ry 0 rz 0.01 deg; joints [30.467, -40.008, 94.856, -144.488, 60.837, 161.841] to (-326.64, 112.04, -44.5) mm, rotated rx 180 ry 0 rz 0.01 deg; joints [30.493, -40.311, 95.506, -144.572, 61.127, 162.057]
  MoveC 4994 to (-320.88, 109.03, -44.5) mm, rotated rx -180 ry 0 rz 0.01 deg; joints [30.505, -40.613, 96.154, -144.669, 61.414, 162.28] to (-315.39, 105.55, -44.5) mm, rotated rx 180 ry 0 rz 0.01 deg; joints [30.497, -40.913, 96.799, -144.786, 61.694, 162.511]
  MoveC 4995 to (-301.09, 93.05, -44.5) mm, rotated rx -180 ry 0 rz 0.01 deg; joints [30.367, -41.759, 98.631, -145.224, 62.459, 163.217] to (-289.92, 77.69, -44.5) mm, rotated rx -180 ry 0 rz 0.01 deg; joints [30.084, -42.529, 100.31, -145.792, 63.122, 163.937]
  MoveL 4996 to (-271.17, 44.94, -44.5) mm, rotated rx 180 ry 0 rz 0.01 deg; joints [29.362, -43.929, 103.388, -147.021, 64.312, 165.322]
  MoveC 4997 to (-269.8, 42.33, -44.5) mm, rotated rx 180 ry 0 rz 0.01 deg; joints [29.301, -44.033, 103.618, -147.12, 64.401, 165.427] to (-268.65, 39.61, -44.5) mm, rotated rx -180 ry 0 rz 0.01 deg; joints [29.232, -44.131, 103.835, -147.224, 64.482, 165.531]
  MoveC 4998 to (-267.6, 36.86, -44.5) mm, rotated rx 180 ry 0 rz 0.01 deg; joints [29.16, -44.226, 104.046, -147.331, 64.56, 165.634] to (-266.49, 34.13, -44.5) mm, rotated rx -180 ry 0 rz 0.01 deg; joints [29.089, -44.322, 104.259, -147.436, 64.639, 165.737]
  MoveC 4999 to (-264.01, 31.11, -44.5) mm, rotated rx 180 ry 0 rz 0.01 deg; joints [29.034, -44.475, 104.596, -147.542, 64.78, 165.872] to (-260.27, 29.97, -44.5) mm, rotated rx 180 ry 0 rz 0.01 deg; joints [29.066, -44.637, 104.949, -147.556, 64.95, 165.971]
  MoveL 5000 to (-133.26, 29.97, -44.5) mm, rotated rx -180 ry 0 rz 0.01 deg; joints [31.633, -49.083, 114.701, -146.066, 70.028, 168.056]
  MoveC 5001 to (-129.5, 31.11, -44.5) mm, rotated rx -180 ry 0 rz 0.01 deg; joints [31.755, -49.184, 114.924, -145.964, 70.157, 168.084] to (-127.01, 34.13, -44.5) mm, rotated rx -180 ry 0 rz 0.01 deg; joints [31.917, -49.207, 114.969, -145.801, 70.213, 168.038]
  MoveC 5002 to (-125.85, 36.97, -44.5) mm, rotated rx 180 ry 0 rz 0.01 deg; joints [32.043, -49.19, 114.924, -145.665, 70.219, 167.976] to (-124.76, 39.83, -44.5) mm, rotated rx -180 ry 0 rz 0.01 deg; joints [32.169, -49.17, 114.874, -145.529, 70.223, 167.913]
  MoveC 5003 to (-123.57, 42.66, -44.5) mm, rotated rx -180 ry 0 rz 0.01 deg; joints [32.295, -49.153, 114.831, -145.394, 70.231, 167.852] to (-122.14, 45.38, -44.5) mm, rotated rx -180 ry 0 rz 0.01 deg; joints [32.422, -49.146, 114.809, -145.259, 70.249, 167.797]
  MoveL 5004 to (-103.04, 78.44, -44.5) mm, rotated rx 180 ry 0 rz 0.01 deg; joints [34.008, -49.097, 114.63, -143.598, 70.524, 167.151]
  MoveC 5005 to (-91.42, 94.08, -44.5) mm, rotated rx 180 ry 0 rz 0.01 deg; joints [34.818, -49.141, 114.696, -142.771, 70.743, 166.88] to (-76.54, 106.66, -44.5) mm, rotated rx 180 ry 0 rz 0.01 deg; joints [35.603, -49.342, 115.117, -142.013, 71.115, 166.751]
  MoveC 5006 to (-71.4, 109.78, -44.5) mm, rotated rx 180 ry 0 rz 0.01 deg; joints [35.834, -49.436, 115.319, -141.8, 71.258, 166.743] to (-66.02, 112.46, -44.5) mm, rotated rx 180 ry 0 rz 0.01 deg; joints [36.058, -49.545, 115.557, -141.599, 71.416, 166.752]
  MoveC 5007 to (-60.5, 114.86, -44.5) mm, rotated rx -180 ry 0 rz 0.01 deg; joints [36.275, -49.664, 115.816, -141.406, 71.581, 166.771] to (-54.95, 117.15, -44.5) mm, rotated rx 180 ry 0 rz 0.01 deg; joints [36.491, -49.785, 116.082, -141.216, 71.748, 166.795]
  MoveC 5008 to (-52.06, 119.47, -44.5) mm, rotated rx -180 ry 0 rz 0.01 deg; joints [36.643, -49.823, 116.162, -141.07, 71.819, 166.773] to (-50.97, 123.02, -44.5) mm, rotated rx 180 ry 0 rz 0.01 deg; joints [36.79, -49.779, 116.056, -140.908, 71.808, 166.684]
  MoveL 5009 to (-50.97, 274.12, -44.5) mm, rotated rx 180 ry 0 rz 0.01 deg; joints [41.553, -46.107, 107.697, -134.987, 69.731, 161.715]
  MoveC 5010 to (-52.1, 276.84, -44.5) mm, rotated rx -180 ry 0 rz 0.01 deg; joints [41.604, -45.999, 107.458, -134.902, 69.655, 161.598] to (-54.82, 277.97, -44.5) mm, rotated rx -180 ry 0 rz 0.01 deg; joints [41.566, -45.884, 107.205, -134.904, 69.546, 161.508]
  MoveL 5011 to (-84.5, 277.97, -44.5) mm, rotated rx -180 ry 0 rz 0.01 deg; joints [40.806, -44.943, 105.164, -135.37, 68.504, 160.958]
  MoveC 5012 to (-87.75, 276.84, -44.5) mm, rotated rx -180 ry 0 rz 0.01 deg; joints [40.691, -44.868, 105.004, -135.462, 68.403, 160.938] to (-89.61, 273.92, -44.5) mm, rotated rx 180 ry 0 rz 0.01 deg; joints [40.559, -44.887, 105.049, -135.602, 68.376, 161.008]
  MoveC 5013 to (-106.66, 239.26, -44.5) mm, rotated rx -180 ry 0 rz 0.01 deg; joints [39.108, -45.246, 105.884, -137.202, 68.226, 161.92] to (-137.08, 215.46, -44.5) mm, rotated rx -180 ry 0 rz 0.01 deg; joints [37.655, -44.841, 105.048, -138.564, 67.425, 162.182]
  MoveC 5014 to (-147.02, 211.35, -44.5) mm, rotated rx -180 ry 0 rz 0.01 deg; joints [37.297, -44.607, 104.549, -138.857, 67.108, 162.138] to (-157.3, 208.23, -44.5) mm, rotated rx 180 ry 0 rz 0.01 deg; joints [36.964, -44.334, 103.963, -139.112, 66.762, 162.052]
  MoveC 5015 to (-167.88, 206.25, -44.5) mm, rotated rx -180 ry 0 rz 0.01 deg; joints [36.661, -44.017, 103.283, -139.32, 66.387, 161.921] to (-178.62, 205.58, -44.5) mm, rotated rx 180 ry 0 rz 0.01 deg; joints [36.399, -43.658, 102.51, -139.472, 65.985, 161.738]
  MoveL 5016 to (-216.07, 205.58, -44.5) mm, rotated rx -180 ry 0 rz 0.01 deg; joints [35.574, -42.313, 99.62, -139.864, 64.525, 161.004]
  MoveC 5017 to (-235.57, 207.8, -44.5) mm, rotated rx -180 ry 0 rz 0.01 deg; joints [35.223, -41.533, 97.949, -139.95, 63.72, 160.528] to (-254.09, 214.32, -44.5) mm, rotated rx 180 ry 0 rz 0.01 deg; joints [35.029, -40.663, 96.082, -139.83, 62.887, 159.902]
  MoveC 5018 to (-268.37, 222.8, -44.5) mm, rotated rx -180 ry 0 rz 0.01 deg; joints [34.984, -39.887, 94.418, -139.579, 62.193, 159.277] to (-281.02, 233.55, -44.5) mm, rotated rx 180 ry 0 rz 0.01 deg; joints [35.039, -39.1, 92.73, -139.207, 61.53, 158.584]
  MoveC 5019 to (-283.06, 237.54, -44.5) mm, rotated rx -180 ry 0 rz 0.01 deg; joints [35.114, -38.91, 92.321, -139.051, 61.393, 158.384] to (-282.42, 241.97, -44.5) mm, rotated rx 180 ry 0 rz 0.01 deg; joints [35.255, -38.815, 92.112, -138.862, 61.363, 158.226]
  MoveC 5020 to (-281.6, 246.32, -44.5) mm, rotated rx 180 ry 0 rz 0.01 deg; joints [35.397, -38.728, 91.921, -138.676, 61.341, 158.075] to (-283.11, 250.48, -44.5) mm, rotated rx 180 ry 0 rz 0.01 deg; joints [35.486, -38.552, 91.542, -138.509, 61.224, 157.876]
  MoveC 5021 to (-285.5, 254.01, -44.5) mm, rotated rx -180 ry 0 rz 0.01 deg; joints [35.538, -38.358, 91.125, -138.374, 61.078, 157.681] to (-287.75, 257.62, -44.5) mm, rotated rx 180 ry 0 rz 0.01 deg; joints [35.595, -38.165, 90.713, -138.233, 60.937, 157.484]
  MoveC 5022 to (-291.88, 265.86, -44.5) mm, rotated rx 180 ry 0 rz 0.01 deg; joints [35.746, -37.764, 89.853, -137.904, 60.657, 157.054] to (-294.73, 274.62, -44.5) mm, rotated rx -180 ry 0 rz 0.01 deg; joints [35.935, -37.395, 89.061, -137.546, 60.423, 156.628]
  MoveC 5023 to (-295.22, 276.78, -44.5) mm, rotated rx 180 ry 0 rz 0.01 deg; joints [35.986, -37.312, 88.883, -137.456, 60.374, 156.528] to (-295.63, 278.95, -44.5) mm, rotated rx -180 ry 0 rz 0.01 deg; joints [36.038, -37.232, 88.711, -137.366, 60.328, 156.428]
  MoveC 5024 to (-296.03, 281.13, -44.5) mm, rotated rx 180 ry 0 rz 0.01 deg; joints [36.091, -37.152, 88.538, -137.275, 60.283, 156.328] to (-296.48, 283.3, -44.5) mm, rotated rx 180 ry 0 rz 0.01 deg; joints [36.143, -37.07, 88.362, -137.185, 60.235, 156.227]
  MoveC 5025 to (-298.29, 286.19, -44.5) mm, rotated rx -180 ry 0 rz 0.01 deg; joints [36.187, -36.909, 88.02, -137.068, 60.121, 156.061] to (-301.51, 287.33, -44.5) mm, rotated rx 180 ry 0 rz 0.01 deg; joints [36.153, -36.742, 87.666, -137.03, 59.97, 155.933]
  MoveL 5026 to (-348.06, 287.33, -44.5) mm, rotated rx -180 ry 0 rz 0.01 deg; joints [35.226, -34.742, 83.465, -137.099, 57.951, 154.693]
  MoveC 5027 to (-350.78, 286.2, -44.5) mm, rotated rx 180 ry 0 rz 0.01 deg; joints [35.142, -34.656, 83.285, -137.148, 57.845, 154.667] to (-351.91, 283.47, -44.5) mm, rotated rx -180 ry 0 rz 0.01 deg; joints [35.045, -34.689, 83.358, -137.267, 57.831, 154.754]
  MoveL 5028 to (-351.91, 115.52, -44.5) mm, rotated rx -180 ry 0 rz 0.01 deg; joints [30.143, -39.19, 93.116, -144.535, 59.976, 161.402]
  MoveC 5029 to (-350.82, 112.32, -44.5) mm, rotated rx -180 ry 0 rz 0.01 deg; joints [30.064, -39.31, 93.377, -144.668, 60.064, 161.54] to (-348, 110.45, -44.5) mm, rotated rx -180 ry 0 rz 0.01 deg; joints [30.056, -39.471, 93.721, -144.737, 60.211, 161.666]
  MoveC 5030 to (-338.2, 107.18, -44.5) mm, rotated rx 180 ry 0 rz 0.01 deg; joints [30.131, -39.951, 94.748, -144.835, 60.683, 161.988] to (-328.87, 102.72, -44.5) mm, rotated rx -180 ry 0 rz 0.01 deg; joints [30.161, -40.434, 95.783, -144.979, 61.145, 162.335]
  MoveC 5031 to (-320.14, 97.18, -44.5) mm, rotated rx -180 ry 0 rz 0.01 deg; joints [30.146, -40.911, 96.81, -145.167, 61.591, 162.702] to (-312.12, 90.66, -44.5) mm, rotated rx -180 ry 0 rz 0.01 deg; joints [30.087, -41.376, 97.816, -145.395, 62.017, 163.082]
  MoveC 5032 to (-307.86, 86.42, -44.5) mm, rotated rx -180 ry 0 rz 0.01 deg; joints [30.031, -41.638, 98.385, -145.548, 62.252, 163.307] to (-303.97, 81.82, -44.5) mm, rotated rx -180 ry 0 rz 0.01 deg; joints [29.956, -41.892, 98.936, -145.717, 62.474, 163.535]
  MoveC 5033 to (-300.45, 76.94, -44.5) mm, rotated rx -180 ry 0 rz 0.01 deg; joints [29.864, -42.136, 99.468, -145.899, 62.684, 163.764] to (-297.27, 71.83, -44.5) mm, rotated rx -180 ry 0 rz 0.01 deg; joints [29.758, -42.369, 99.978, -146.092, 62.882, 163.991]
  MoveL 5034 to (-283.34, 47.66, -44.5) mm, rotated rx -180 ry 0 rz 0.01 deg; joints [29.226, -43.412, 102.266, -147.006, 63.767, 165.021]
  MoveC 5035 to (-277.5, 36.35, -44.5) mm, rotated rx -180 ry 0 rz 0.01 deg; joints [28.959, -43.863, 103.261, -147.436, 64.15, 165.477] to (-272.75, 24.55, -44.5) mm, rotated rx -180 ry 0 rz 0.01 deg; joints [28.652, -44.276, 104.179, -147.894, 64.493, 165.922]
  MoveC 5036 to (-270.6, 21.69, -44.5) mm, rotated rx -180 ry 0 rz 0.01 deg; joints [28.595, -44.413, 104.48, -147.996, 64.617, 166.045] to (-267.2, 20.61, -44.5) mm, rotated rx 180 ry 0 rz 0.01 deg; joints [28.621, -44.562, 104.804, -148.012, 64.773, 166.136]
  MoveL 5037 to (-126.31, 20.61, -44.5) mm, rotated rx 180 ry 0 rz 0.01 deg; joints [31.452, -49.489, 115.626, -146.357, 70.419, 168.428]
  MoveC 5038 to (-122.91, 21.69, -44.5) mm, rotated rx -180 ry 0 rz 0.01 deg; joints [31.565, -49.579, 115.825, -146.261, 70.534, 168.452] to (-120.76, 24.55, -44.5) mm, rotated rx -180 ry 0 rz 0.01 deg; joints [31.714, -49.595, 115.854, -146.11, 70.579, 168.406]
  MoveC 5039 to (-115.94, 36.52, -44.5) mm, rotated rx -180 ry 0 rz 0.01 deg; joints [32.248, -49.521, 115.663, -145.536, 70.603, 168.148] to (-110.01, 47.99, -44.5) mm, rotated rx -180 ry 0 rz 0.01 deg; joints [32.787, -49.488, 115.565, -144.967, 70.674, 167.918]
  MoveL 5040 to (-96.03, 72.18, -44.5) mm, rotated rx 180 ry 0 rz 0.01 deg; joints [33.955, -49.45, 115.428, -143.745, 70.87, 167.449]
  MoveC 5041 to (-90.46, 80.53, -44.5) mm, rotated rx -180 ry 0 rz 0.01 deg; joints [34.375, -49.455, 115.421, -143.311, 70.963, 167.296] to (-83.87, 88.1, -44.5) mm, rotated rx 180 ry 0 rz 0.01 deg; joints [34.793, -49.506, 115.519, -142.893, 71.102, 167.182]
  MoveC 5042 to (-76.45, 94.86, -44.5) mm, rotated rx 180 ry 0 rz 0.01 deg; joints [35.203, -49.596, 115.707, -142.493, 71.28, 167.104] to (-68.39, 100.83, -44.5) mm, rotated rx 180 ry 0 rz 0.01 deg; joints [35.604, -49.721, 115.972, -142.112, 71.491, 167.06]
  MoveC 5043 to (-63.02, 104, -44.5) mm, rotated rx -180 ry 0 rz 0.01 deg; joints [35.844, -49.82, 116.187, -141.89, 71.641, 167.055] to (-57.34, 106.56, -44.5) mm, rotated rx -180 ry 0 rz 0.01 deg; joints [36.072, -49.94, 116.45, -141.687, 71.81, 167.073]
  MoveC 5044 to (-51.47, 108.66, -44.5) mm, rotated rx 180 ry 0 rz 0.01 deg; joints [36.29, -50.075, 116.747, -141.498, 71.99, 167.107] to (-45.51, 110.45, -44.5) mm, rotated rx 180 ry 0 rz 0.01 deg; joints [36.501, -50.218, 117.063, -141.317, 72.178, 167.152]
  MoveC 5045 to (-42.69, 112.35, -44.5) mm, rotated rx 180 ry 0 rz 0.01 deg; joints [36.637, -50.263, 117.159, -141.189, 72.251, 167.142] to (-41.6, 115.56, -44.5) mm, rotated rx -180 ry 0 rz 0.01 deg; joints [36.774, -50.226, 117.071, -141.039, 72.245, 167.064]
  MoveL 5046 to (-41.61, 283.48, -44.5) mm, rotated rx 180 ry 0 rz 0.01 deg; joints [42.073, -46.145, 107.765, -134.473, 69.927, 161.552]
  MoveC 5047 to (-42.74, 286.2, -44.5) mm, rotated rx 180 ry 0 rz 0.01 deg; joints [42.123, -46.037, 107.524, -134.389, 69.852, 161.434] to (-45.46, 287.33, -44.5) mm, rotated rx -180 ry 0 rz 0.01 deg; joints [42.084, -45.922, 107.272, -134.392, 69.743, 161.344]
  MoveL 5048 to (-91.95, 287.33, -44.5) mm, rotated rx 180 ry 0 rz 0.01 deg; joints [40.891, -44.447, 104.076, -135.119, 68.114, 160.477]
  MoveC 5049 to (-95.17, 286.21, -44.5) mm, rotated rx -180 ry 0 rz 0.01 deg; joints [40.778, -44.372, 103.917, -135.209, 68.013, 160.457] to (-97, 283.33, -44.5) mm, rotated rx -180 ry 0 rz 0.01 deg; joints [40.649, -44.391, 103.962, -135.346, 67.986, 160.527]
  MoveL 5050 to (-99.84, 271.34, -44.5) mm, rotated rx -180 ry 0 rz 0.01 deg; joints [40.228, -44.623, 104.483, -135.852, 68.044, 160.908]
  MoveC 5051 to (-101.57, 265.78, -44.5) mm, rotated rx -180 ry 0 rz 0.01 deg; joints [40.022, -44.716, 104.692, -136.093, 68.056, 161.075] to (-104.06, 260.51, -44.5) mm, rotated rx 180 ry 0 rz 0.01 deg; joints [39.805, -44.774, 104.827, -136.334, 68.036, 161.217]
  MoveC 5052 to (-117.58, 242.14, -44.5) mm, rotated rx -180 ry 0 rz 0.01 deg; joints [38.928, -44.811, 104.937, -137.244, 67.79, 161.615] to (-135.16, 227.62, -44.5) mm, rotated rx -180 ry 0 rz 0.01 deg; joints [38.07, -44.597, 104.499, -138.055, 67.335, 161.794]
  MoveC 5053 to (-155.98, 218.18, -44.5) mm, rotated rx 180 ry 0 rz 0.01 deg; joints [37.297, -44.128, 103.502, -138.697, 66.681, 161.731] to (-178.62, 214.95, -44.5) mm, rotated rx 180 ry 0 rz 0.01 deg; joints [36.683, -43.421, 101.985, -139.095, 65.862, 161.409]
  MoveL 5054 to (-222.09, 215.41, -44.5) mm, rotated rx 180 ry 0 rz 0.01 deg; joints [35.739, -41.839, 98.591, -139.52, 64.159, 160.528]
  MoveC 5055 to (-237.42, 218.56, -44.5) mm, rotated rx 180 ry 0 rz 0.01 deg; joints [35.505, -41.186, 97.189, -139.524, 63.506, 160.097] to (-252.13, 223.91, -44.5) mm, rotated rx 180 ry 0 rz 0.01 deg; joints [35.354, -40.487, 95.69, -139.419, 62.843, 159.588]
  MoveC 5056 to (-265.65, 231.9, -44.5) mm, rotated rx 180 ry 0 rz 0.01 deg; joints [35.307, -39.751, 94.113, -139.183, 62.187, 158.992] to (-277.07, 242.68, -44.5) mm, rotated rx 180 ry 0 rz 0.01 deg; joints [35.385, -39.008, 92.521, -138.803, 61.576, 158.321]
  MoveC 5057 to (-280.17, 246.52, -44.5) mm, rotated rx 180 ry 0 rz 0.01 deg; joints [35.432, -38.779, 92.03, -138.66, 61.398, 158.1] to (-283.11, 250.48, -44.5) mm, rotated rx -180 ry 0 rz 0.01 deg; joints [35.486, -38.552, 91.542, -138.509, 61.224, 157.876]
  MoveC 5058 to (-284.53, 254.91, -44.5) mm, rotated rx -180 ry 0 rz 0.01 deg; joints [35.584, -38.371, 91.153, -138.331, 61.107, 157.668] to (-283.17, 259.36, -44.5) mm, rotated rx -180 ry 0 rz 0.01 deg; joints [35.739, -38.301, 90.998, -138.138, 61.106, 157.523]
  MoveC 5059 to (-281.62, 263.68, -44.5) mm, rotated rx -180 ry 0 rz 0.01 deg; joints [35.894, -38.241, 90.865, -137.949, 61.114, 157.387] to (-282.39, 268.2, -44.5) mm, rotated rx -180 ry 0 rz 0.01 deg; joints [36.007, -38.082, 90.52, -137.763, 61.023, 157.188]
  MoveC 5060 to (-284.98, 274.8, -44.5) mm, rotated rx -180 ry 0 rz 0.01 deg; joints [36.14, -37.787, 89.889, -137.497, 60.829, 156.858] to (-286.88, 281.64, -44.5) mm, rotated rx -180 ry 0 rz 0.01 deg; joints [36.293, -37.512, 89.297, -137.218, 60.661, 156.533]
  MoveC 5061 to (-287.97, 287.24, -44.5) mm, rotated rx -180 ry 0 rz 0.01 deg; joints [36.427, -37.303, 88.848, -136.986, 60.542, 156.276] to (-288.75, 292.89, -44.5) mm, rotated rx -180 ry 0 rz 0.01 deg; joints [36.569, -37.104, 88.42, -136.75, 60.435, 156.022]
  MoveC 5062 to (-290.15, 295.6, -44.5) mm, rotated rx 180 ry 0 rz 0.01 deg; joints [36.615, -36.966, 88.125, -136.641, 60.341, 155.874] to (-292.99, 296.69, -44.5) mm, rotated rx 180 ry 0 rz 0.01 deg; joints [36.587, -36.816, 87.808, -136.605, 60.207, 155.756]
  MoveL 5063 to (-357.42, 296.69, -44.5) mm, rotated rx 180 ry 0 rz 0.01 deg; joints [35.301, -34.034, 81.967, -136.679, 57.409, 154.012]
  MoveC 5064 to (-360.14, 295.56, -44.5) mm, rotated rx 180 ry 0 rz 0.01 deg; joints [35.218, -33.946, 81.784, -136.725, 57.302, 153.983] to (-361.27, 292.83, -44.5) mm, rotated rx 180 ry 0 rz 0.01 deg; joints [35.122, -33.98, 81.859, -136.845, 57.287, 154.073]
  MoveL 5065 to (-361.27, 107.6, -44.5) mm, rotated rx 180 ry 0 rz 0.01 deg; joints [29.733, -38.982, 92.687, -144.907, 59.657, 161.483]
  MoveC 5066 to (-360.14, 104.48, -44.5) mm, rotated rx -180 ry 0 rz 0.01 deg; joints [29.656, -39.101, 92.947, -145.037, 59.745, 161.619] to (-357.27, 102.8, -44.5) mm, rotated rx -180 ry 0 rz 0.01 deg; joints [29.655, -39.261, 93.287, -145.099, 59.893, 161.74]
  MoveL 5067 to (-350.13, 101.48, -44.5) mm, rotated rx 180 ry 0 rz 0.01 deg; joints [29.74, -39.589, 93.988, -145.129, 60.227, 161.938]
  MoveC 5068 to (-346.79, 100.67, -44.5) mm, rotated rx -180 ry 0 rz 0.01 deg; joints [29.774, -39.746, 94.323, -145.15, 60.385, 162.037] to (-343.57, 99.47, -44.5) mm, rotated rx -180 ry 0 rz 0.01 deg; joints [29.794, -39.906, 94.666, -145.187, 60.541, 162.146]
  MoveC 5069 to (-332.3, 93.62, -44.5) mm, rotated rx -180 ry 0 rz 0.01 deg; joints [29.813, -40.499, 95.939, -145.383, 61.107, 162.579] to (-321.89, 86.37, -44.5) mm, rotated rx 180 ry 0 rz 0.01 deg; joints [29.773, -41.081, 97.194, -145.635, 61.648, 163.035]
  MoveC 5070 to (-312.73, 77.54, -44.5) mm, rotated rx 180 ry 0 rz 0.01 deg; joints [29.658, -41.639, 98.403, -145.954, 62.151, 163.509] to (-305.38, 67.16, -44.5) mm, rotated rx 180 ry 0 rz 0.01 deg; joints [29.458, -42.152, 99.521, -146.345, 62.593, 163.991]
  MoveC 5071 to (-298.05, 54.65, -44.5) mm, rotated rx -180 ry 0 rz 0.01 deg; joints [29.186, -42.701, 100.723, -146.822, 63.058, 164.532] to (-290.53, 42.25, -44.5) mm, rotated rx -180 ry 0 rz 0.01 deg; joints [28.916, -43.246, 101.92, -147.29, 63.528, 165.062]
  MoveC 5072 to (-284.02, 29.23, -44.5) mm, rotated rx -180 ry 0 rz 0.01 deg; joints [28.602, -43.757, 103.047, -147.789, 63.961, 165.583] to (-279.9, 15.26, -44.5) mm, rotated rx 180 ry 0 rz 0.01 deg; joints [28.209, -44.187, 104.004, -148.346, 64.303, 166.081]
  MoveC 5073 to (-278.16, 12.38, -44.5) mm, rotated rx 180 ry 0 rz 0.01 deg; joints [28.143, -44.309, 104.273, -148.454, 64.411, 166.198] to (-274.99, 11.25, -44.5) mm, rotated rx 180 ry 0 rz 0.01 deg; joints [28.162, -44.45, 104.581, -148.475, 64.558, 166.286]
  MoveL 5074 to (-118.59, 11.25, -44.5) mm, rotated rx -180 ry 0 rz 0.01 deg; joints [31.284, -49.916, 116.601, -146.637, 70.838, 168.808]
  MoveC 5075 to (-115.39, 12.38, -44.5) mm, rotated rx -180 ry 0 rz 0.01 deg; joints [31.396, -49.999, 116.783, -146.541, 70.946, 168.827] to (-113.62, 15.27, -44.5) mm, rotated rx 180 ry 0 rz 0.01 deg; joints [31.539, -50.002, 116.784, -146.392, 70.975, 168.775]
  MoveC 5076 to (-112.3, 20.67, -44.5) mm, rotated rx 180 ry 0 rz 0.01 deg; joints [31.763, -49.943, 116.639, -146.145, 70.953, 168.648] to (-110.66, 25.98, -44.5) mm, rotated rx 180 ry 0 rz 0.01 deg; joints [31.99, -49.894, 116.52, -145.897, 70.944, 168.526]
  MoveC 5077 to (-108.61, 31.15, -44.5) mm, rotated rx -180 ry 0 rz 0.01 deg; joints [32.221, -49.861, 116.434, -145.648, 70.952, 168.415] to (-106.07, 36.09, -44.5) mm, rotated rx 180 ry 0 rz 0.01 deg; joints [32.455, -49.847, 116.392, -145.402, 70.982, 168.317]
  MoveL 5078 to (-84.51, 72.59, -44.5) mm, rotated rx -180 ry 0 rz 0.01 deg; joints [34.24, -49.806, 116.221, -143.541, 71.29, 167.625]
  MoveC 5079 to (-75.25, 82.91, -44.5) mm, rotated rx 180 ry 0 rz 0.01 deg; joints [34.82, -49.884, 116.373, -142.962, 71.488, 167.476] to (-64.56, 91.74, -44.5) mm, rotated rx 180 ry 0 rz 0.01 deg; joints [35.385, -50.032, 116.686, -142.417, 71.755, 167.392]
  MoveC 5080 to (-52.39, 98.48, -44.5) mm, rotated rx 180 ry 0 rz 0.01 deg; joints [35.918, -50.264, 117.191, -141.927, 72.1, 167.394] to (-39.04, 102.41, -44.5) mm, rotated rx 180 ry 0 rz 0.01 deg; joints [36.389, -50.586, 117.904, -141.525, 72.521, 167.498]
  MoveC 5081 to (-38.34, 102.52, -44.5) mm, rotated rx 180 ry 0 rz 0.01 deg; joints [36.411, -50.605, 117.946, -141.508, 72.544, 167.506] to (-37.64, 102.62, -44.5) mm, rotated rx 180 ry 0 rz 0.01 deg; joints [36.432, -50.624, 117.989, -141.491, 72.568, 167.515]
  MoveC 5082 to (-36.94, 102.71, -44.5) mm, rotated rx -180 ry 0 rz 0.01 deg; joints [36.453, -50.643, 118.032, -141.474, 72.591, 167.524] to (-36.24, 102.82, -44.5) mm, rotated rx 180 ry 0 rz 0.01 deg; joints [36.475, -50.662, 118.074, -141.457, 72.614, 167.532]
  MoveC 5083 to (-33.37, 104.48, -44.5) mm, rotated rx 180 ry 0 rz 0.01 deg; joints [36.605, -50.712, 118.184, -141.336, 72.692, 167.53] to (-32.24, 107.59, -44.5) mm, rotated rx 180 ry 0 rz 0.01 deg; joints [36.741, -50.68, 118.104, -141.188, 72.688, 167.457]
  MoveL 5084 to (-32.25, 292.84, -44.5) mm, rotated rx -180 ry 0 rz 0.01 deg; joints [42.594, -46.178, 107.821, -133.959, 70.121, 161.387]
  MoveC 5085 to (-33.37, 295.57, -44.5) mm, rotated rx 180 ry 0 rz 0.01 deg; joints [42.642, -46.069, 107.579, -133.876, 70.046, 161.268] to (-36.1, 296.7, -44.5) mm, rotated rx -180 ry 0 rz 0.01 deg; joints [42.603, -45.955, 107.329, -133.88, 69.938, 161.177]
  MoveL 5086 to (-100.55, 296.69, -44.5) mm, rotated rx 180 ry 0 rz 0.01 deg; joints [40.946, -43.906, 102.896, -134.88, 67.681, 159.967]
  MoveC 5087 to (-103.38, 295.61, -44.5) mm, rotated rx 180 ry 0 rz 0.01 deg; joints [40.844, -43.843, 102.762, -134.961, 67.594, 159.953] to (-104.75, 292.9, -44.5) mm, rotated rx -180 ry 0 rz 0.01 deg; joints [40.733, -43.873, 102.83, -135.085, 67.58, 160.026]
  MoveC 5088 to (-106.06, 284.39, -44.5) mm, rotated rx 180 ry 0 rz 0.01 deg; joints [40.455, -44.064, 103.256, -135.433, 67.646, 160.315] to (-108.18, 276.05, -44.5) mm, rotated rx -180 ry 0 rz 0.01 deg; joints [40.16, -44.222, 103.608, -135.787, 67.68, 160.579]
  MoveC 5089 to (-111.15, 267.96, -44.5) mm, rotated rx -180 ry 0 rz 0.01 deg; joints [39.851, -44.342, 103.88, -136.143, 67.681, 160.815] to (-114.95, 260.24, -44.5) mm, rotated rx -180 ry 0 rz 0.01 deg; joints [39.53, -44.422, 104.066, -136.498, 67.645, 161.021]
  MoveC 5090 to (-122.92, 249.06, -44.5) mm, rotated rx 180 ry 0 rz 0.01 deg; joints [39.006, -44.452, 104.15, -137.045, 67.502, 161.269] to (-133.09, 239.85, -44.5) mm, rotated rx -180 ry 0 rz 0.01 deg; joints [38.487, -44.351, 103.947, -137.544, 67.25, 161.403]
  MoveC 5091 to (-144.76, 232.7, -44.5) mm, rotated rx -180 ry 0 rz 0.01 deg; joints [37.997, -44.141, 103.505, -137.978, 66.911, 161.434] to (-157.41, 227.47, -44.5) mm, rotated rx 180 ry 0 rz 0.01 deg; joints [37.545, -43.841, 102.868, -138.344, 66.505, 161.377]
  MoveC 5092 to (-162.6, 226.03, -44.5) mm, rotated rx 180 ry 0 rz 0.01 deg; joints [37.382, -43.698, 102.563, -138.464, 66.328, 161.327] to (-167.89, 225.06, -44.5) mm, rotated rx 180 ry 0 rz 0.01 deg; joints [37.231, -43.539, 102.221, -138.565, 66.14, 161.26]
  MoveC 5093 to (-173.24, 224.5, -44.5) mm, rotated rx 180 ry 0 rz 0.01 deg; joints [37.093, -43.366, 101.85, -138.65, 65.943, 161.176] to (-178.62, 224.31, -44.5) mm, rotated rx -180 ry 0 rz 0.01 deg; joints [36.965, -43.182, 101.453, -138.718, 65.74, 161.077]
  MoveL 5094 to (-220.88, 224.7, -44.5) mm, rotated rx 180 ry 0 rz 0.01 deg; joints [36.042, -41.643, 98.156, -139.13, 64.087, 160.215]
  MoveC 5095 to (-234.53, 227.47, -44.5) mm, rotated rx -180 ry 0 rz 0.01 deg; joints [35.831, -41.061, 96.909, -139.135, 63.507, 159.829] to (-247.65, 232.13, -44.5) mm, rotated rx -180 ry 0 rz 0.01 deg; joints [35.69, -40.44, 95.577, -139.047, 62.918, 159.376]
  MoveC 5096 to (-259.74, 239.16, -44.5) mm, rotated rx -180 ry 0 rz 0.01 deg; joints [35.642, -39.785, 94.174, -138.842, 62.336, 158.846] to (-269.93, 248.73, -44.5) mm, rotated rx -180 ry 0 rz 0.01 deg; joints [35.707, -39.125, 92.758, -138.509, 61.793, 158.248]
  MoveC 5097 to (-275.57, 256.17, -44.5) mm, rotated rx 180 ry 0 rz 0.01 deg; joints [35.804, -38.695, 91.835, -138.232, 61.463, 157.827] to (-280.4, 264.16, -44.5) mm, rotated rx 180 ry 0 rz 0.01 deg; joints [35.933, -38.277, 90.939, -137.923, 61.159, 157.397]
  MoveC 5098 to (-281.43, 266.16, -44.5) mm, rotated rx -180 ry 0 rz 0.01 deg; joints [35.969, -38.178, 90.728, -137.844, 61.09, 157.292] to (-282.39, 268.2, -44.5) mm, rotated rx -180 ry 0 rz 0.01 deg; joints [36.007, -38.082, 90.52, -137.763, 61.023, 157.188]
  MoveC 5099 to (-282.94, 272.55, -44.5) mm, rotated rx -180 ry 0 rz 0.01 deg; joints [36.118, -37.935, 90.203, -137.583, 60.944, 156.999] to (-280.95, 276.45, -44.5) mm, rotated rx 180 ry 0 rz 0.01 deg; joints [36.27, -37.903, 90.13, -137.41, 60.976, 156.889]
  MoveC 5100 to (-278.77, 280.17, -44.5) mm, rotated rx -180 ry 0 rz 0.01 deg; joints [36.42, -37.883, 90.083, -137.243, 61.018, 156.79] to (-278.56, 284.48, -44.5) mm, rotated rx -180 ry 0 rz 0.01 deg; joints [36.545, -37.767, 89.83, -137.062, 60.97, 156.62]
  MoveC 5101 to (-278.66, 285.02, -44.5) mm, rotated rx -180 ry 0 rz 0.01 deg; joints [36.558, -37.747, 89.787, -137.039, 60.959, 156.595] to (-278.76, 285.57, -44.5) mm, rotated rx 180 ry 0 rz 0.01 deg; joints [36.571, -37.727, 89.744, -137.017, 60.948, 156.57]
  MoveC 5102 to (-279.65, 293.97, -44.5) mm, rotated rx 180 ry 0 rz 0.01 deg; joints [36.788, -37.444, 89.135, -136.668, 60.801, 156.203] to (-279.42, 302.42, -44.5) mm, rotated rx -180 ry 0 rz 0.01 deg; joints [37.027, -37.201, 88.611, -136.312, 60.699, 155.857]
  MoveC 5103 to (-280.28, 304.97, -44.5) mm, rotated rx 180 ry 0 rz 0.01 deg; joints [37.08, -37.09, 88.372, -136.208, 60.63, 155.729] to (-282.74, 306.05, -44.5) mm, rotated rx 180 ry 0 rz 0.01 deg; joints [37.058, -36.957, 88.09, -136.172, 60.513, 155.622]
  MoveL 5104 to (-366.78, 306.05, -44.5) mm, rotated rx -180 ry 0 rz 0.01 deg; joints [35.375, -33.311, 80.441, -136.243, 56.861, 153.311]
  MoveC 5105 to (-369.51, 304.92, -44.5) mm, rotated rx 180 ry 0 rz 0.01 deg; joints [35.293, -33.221, 80.256, -136.287, 56.753, 153.28] to (-370.64, 302.2, -44.5) mm, rotated rx -180 ry 0 rz 0.01 deg; joints [35.197, -33.256, 80.332, -136.407, 56.738, 153.371]
  MoveL 5106 to (-370.63, 98.48, -44.5) mm, rotated rx -180 ry 0 rz 0.01 deg; joints [29.287, -38.796, 92.309, -145.328, 59.348, 161.607]
  MoveC 5107 to (-369.54, 95.8, -44.5) mm, rotated rx -180 ry 0 rz 0.01 deg; joints [29.223, -38.904, 92.542, -145.441, 59.429, 161.726] to (-366.89, 94.63, -44.5) mm, rotated rx 180 ry 0 rz 0.01 deg; joints [29.233, -39.043, 92.839, -145.483, 59.563, 161.825]
  MoveC 5108 to (-355.32, 93.16, -44.5) mm, rotated rx 180 ry 0 rz 0.01 deg; joints [29.39, -39.562, 93.945, -145.505, 60.098, 162.122] to (-344.23, 89.52, -44.5) mm, rotated rx 180 ry 0 rz 0.01 deg; joints [29.471, -40.104, 95.103, -145.614, 60.633, 162.478]
  MoveC 5109 to (-333.98, 83.99, -44.5) mm, rotated rx -180 ry 0 rz 0.01 deg; joints [29.48, -40.646, 96.269, -145.801, 61.151, 162.875] to (-324.76, 76.85, -44.5) mm, rotated rx -180 ry 0 rz 0.01 deg; joints [29.418, -41.174, 97.41, -146.055, 61.639, 163.299]
  MoveC 5110 to (-321.52, 73.61, -44.5) mm, rotated rx 180 ry 0 rz 0.01 deg; joints [29.373, -41.374, 97.843, -146.173, 61.819, 163.47] to (-318.58, 70.1, -44.5) mm, rotated rx 180 ry 0 rz 0.01 deg; joints [29.314, -41.568, 98.263, -146.305, 61.989, 163.644]
  MoveC 5111 to (-315.91, 66.38, -44.5) mm, rotated rx 180 ry 0 rz 0.01 deg; joints [29.242, -41.753, 98.667, -146.446, 62.149, 163.818] to (-313.49, 62.49, -44.5) mm, rotated rx 180 ry 0 rz 0.01 deg; joints [29.16, -41.932, 99.057, -146.596, 62.301, 163.991]
  MoveL 5112 to (-293.23, 26.69, -44.5) mm, rotated rx 180 ry 0 rz 0.01 deg; joints [28.351, -43.455, 102.399, -147.968, 63.6, 165.5]
  MoveC 5113 to (-291.3, 21.6, -44.5) mm, rotated rx 180 ry 0 rz 0.01 deg; joints [28.216, -43.629, 102.785, -148.169, 63.743, 165.691] to (-289.69, 16.4, -44.5) mm, rotated rx -180 ry 0 rz 0.01 deg; joints [28.071, -43.792, 103.148, -148.376, 63.873, 165.878]
  MoveC 5114 to (-288.48, 11.1, -44.5) mm, rotated rx 180 ry 0 rz 0.01 deg; joints [27.914, -43.942, 103.481, -148.591, 63.988, 166.06] to (-287.74, 5.7, -44.5) mm, rotated rx 180 ry 0 rz 0.01 deg; joints [27.745, -44.073, 103.776, -148.814, 64.084, 166.236]
  MoveC 5115 to (-286.38, 2.98, -44.5) mm, rotated rx -180 ry 0 rz 0.01 deg; joints [27.677, -44.177, 104.006, -148.919, 64.174, 166.341] to (-283.55, 1.88, -44.5) mm, rotated rx -180 ry 0 rz 0.01 deg; joints [27.69, -44.305, 104.286, -148.942, 64.307, 166.422]
  MoveL 5116 to (-110.01, 1.88, -44.5) mm, rotated rx 180 ry 0 rz 0.01 deg; joints [31.133, -50.366, 117.63, -146.902, 71.291, 169.196]
  MoveC 5117 to (-107.11, 3.01, -44.5) mm, rotated rx 180 ry 0 rz 0.01 deg; joints [31.239, -50.438, 117.791, -146.809, 71.386, 169.211] to (-105.73, 5.81, -44.5) mm, rotated rx 180 ry 0 rz 0.01 deg; joints [31.371, -50.431, 117.768, -146.669, 71.402, 169.156]
  MoveC 5118 to (-104.81, 12.48, -44.5) mm, rotated rx 180 ry 0 rz 0.01 deg; joints [31.634, -50.337, 117.541, -146.373, 71.347, 168.99] to (-103.25, 19.04, -44.5) mm, rotated rx 180 ry 0 rz 0.01 deg; joints [31.907, -50.264, 117.362, -146.073, 71.318, 168.835]
  MoveC 5119 to (-100.98, 25.38, -44.5) mm, rotated rx 180 ry 0 rz 0.01 deg; joints [32.187, -50.216, 117.241, -145.771, 71.318, 168.696] to (-97.96, 31.41, -44.5) mm, rotated rx 180 ry 0 rz 0.01 deg; joints [32.472, -50.197, 117.185, -145.47, 71.35, 168.577]
  MoveL 5120 to (-77.09, 66.88, -44.5) mm, rotated rx 180 ry 0 rz 0.01 deg; joints [34.217, -50.155, 117.014, -143.653, 71.642, 167.91]
  MoveC 5121 to (-69.01, 75.98, -44.5) mm, rotated rx 180 ry 0 rz 0.01 deg; joints [34.73, -50.221, 117.142, -143.14, 71.812, 167.779] to (-59.74, 83.86, -44.5) mm, rotated rx 180 ry 0 rz 0.01 deg; joints [35.23, -50.345, 117.403, -142.655, 72.039, 167.702]
  MoveC 5122 to (-49.14, 89.93, -44.5) mm, rotated rx -180 ry 0 rz 0.01 deg; joints [35.704, -50.543, 117.834, -142.218, 72.336, 167.698] to (-37.44, 93.44, -44.5) mm, rotated rx -180 ry 0 rz 0.01 deg; joints [36.12, -50.824, 118.457, -141.861, 72.704, 167.788]
  MoveC 5123 to (-34.75, 93.88, -44.5) mm, rotated rx 180 ry 0 rz 0.01 deg; joints [36.203, -50.895, 118.618, -141.793, 72.794, 167.819] to (-32.05, 94.23, -44.5) mm, rotated rx -180 ry 0 rz 0.01 deg; joints [36.284, -50.969, 118.782, -141.728, 72.884, 167.853]
  MoveC 5124 to (-29.34, 94.49, -44.5) mm, rotated rx -180 ry 0 rz 0.01 deg; joints [36.363, -51.044, 118.953, -141.666, 72.976, 167.89] to (-26.62, 94.63, -44.5) mm, rotated rx 180 ry 0 rz 0.01 deg; joints [36.437, -51.123, 119.129, -141.609, 73.071, 167.93]
  MoveC 5125 to (-23.97, 95.8, -44.5) mm, rotated rx 180 ry 0 rz 0.01 deg; joints [36.546, -51.177, 119.248, -141.511, 73.147, 167.94] to (-22.88, 98.48, -44.5) mm, rotated rx 180 ry 0 rz 0.01 deg; joints [36.667, -51.153, 119.188, -141.38, 73.147, 167.879]
  MoveL 5126 to (-22.88, 302.21, -44.5) mm, rotated rx 180 ry 0 rz 0.01 deg; joints [43.114, -46.206, 107.866, -133.444, 70.312, 161.219]
  MoveC 5127 to (-24.01, 304.93, -44.5) mm, rotated rx 180 ry 0 rz 0.01 deg; joints [43.162, -46.096, 107.624, -133.361, 70.237, 161.099] to (-26.74, 306.06, -44.5) mm, rotated rx 180 ry 0 rz 0.01 deg; joints [43.121, -45.982, 107.374, -133.366, 70.13, 161.009]
  MoveL 5128 to (-110.81, 306.06, -44.5) mm, rotated rx 180 ry 0 rz 0.01 deg; joints [40.959, -43.304, 101.586, -134.658, 67.187, 159.418]
  MoveC 5129 to (-113.25, 304.96, -44.5) mm, rotated rx 180 ry 0 rz 0.01 deg; joints [40.868, -43.254, 101.478, -134.732, 67.113, 159.411] to (-114.07, 302.41, -44.5) mm, rotated rx 180 ry 0 rz 0.01 deg; joints [40.775, -43.298, 101.578, -134.842, 67.117, 159.491]
  MoveC 5130 to (-115.32, 282.68, -44.5) mm, rotated rx -180 ry 0 rz 0.01 deg; joints [40.178, -43.804, 102.697, -135.626, 67.334, 160.199] to (-123.24, 264.57, -44.5) mm, rotated rx -180 ry 0 rz 0.01 deg; joints [39.457, -44.03, 103.213, -136.44, 67.285, 160.706]
  MoveC 5131 to (-136.25, 249.83, -44.5) mm, rotated rx -180 ry 0 rz 0.01 deg; joints [38.71, -43.983, 103.136, -137.191, 67.001, 160.987] to (-152.73, 239.13, -44.5) mm, rotated rx 180 ry 0 rz 0.01 deg; joints [38.003, -43.7, 102.544, -137.822, 66.527, 161.052]
  MoveC 5132 to (-157.81, 237.12, -44.5) mm, rotated rx 180 ry 0 rz 0.01 deg; joints [37.825, -43.578, 102.284, -137.964, 66.363, 161.026] to (-163.09, 235.74, -44.5) mm, rotated rx -180 ry 0 rz 0.01 deg; joints [37.662, -43.43, 101.969, -138.082, 66.182, 160.972]
  MoveC 5133 to (-168.45, 234.77, -44.5) mm, rotated rx 180 ry 0 rz 0.01 deg; joints [37.51, -43.268, 101.622, -138.183, 65.991, 160.902] to (-173.84, 233.98, -44.5) mm, rotated rx 180 ry 0 rz 0.01 deg; joints [37.363, -43.099, 101.261, -138.276, 65.796, 160.825]
  MoveL 5134 to (-214.9, 233.67, -44.5) mm, rotated rx -180 ry 0 rz 0.01 deg; joints [36.438, -41.628, 98.11, -138.71, 64.207, 160.009]
  MoveC 5135 to (-232.63, 236.25, -44.5) mm, rotated rx 180 ry 0 rz 0.01 deg; joints [36.131, -40.9, 96.55, -138.759, 63.469, 159.542] to (-248.89, 243.78, -44.5) mm, rotated rx 180 ry 0 rz 0.01 deg; joints [36.004, -40.079, 94.792, -138.576, 62.717, 158.908]
  MoveC 5136 to (-262.57, 255.26, -44.5) mm, rotated rx -180 ry 0 rz 0.01 deg; joints [36.049, -39.233, 92.978, -138.193, 62.011, 158.161] to (-273.12, 269.67, -44.5) mm, rotated rx -180 ry 0 rz 0.01 deg; joints [36.24, -38.411, 91.215, -137.654, 61.389, 157.348]
  MoveC 5137 to (-276.43, 276.86, -44.5) mm, rotated rx 180 ry 0 rz 0.01 deg; joints [36.375, -38.073, 90.489, -137.371, 61.158, 156.981] to (-278.56, 284.48, -44.5) mm, rotated rx 180 ry 0 rz 0.01 deg; joints [36.545, -37.767, 89.83, -137.062, 60.97, 156.62]
  MoveC 5138 to (-278.09, 288.86, -44.5) mm, rotated rx 180 ry 0 rz 0.01 deg; joints [36.677, -37.657, 89.593, -136.876, 60.932, 156.452] to (-275.25, 292.22, -44.5) mm, rotated rx 180 ry 0 rz 0.01 deg; joints [36.831, -37.673, 89.622, -136.722, 61.007, 156.383]
  MoveC 5139 to (-272.24, 295.33, -44.5) mm, rotated rx -180 ry 0 rz 0.01 deg; joints [36.981, -37.703, 89.679, -136.577, 61.09, 156.328] to (-270.97, 299.46, -44.5) mm, rotated rx -180 ry 0 rz 0.01 deg; joints [37.122, -37.631, 89.522, -136.398, 61.089, 156.189]
  MoveL 5140 to (-270.9, 300.37, -44.5) mm, rotated rx -180 ry 0 rz 0.01 deg; joints [37.149, -37.607, 89.47, -136.36, 61.079, 156.153]
  MoveC 5141 to (-270.56, 303.15, -44.5) mm, rotated rx -180 ry 0 rz 0.01 deg; joints [37.233, -37.538, 89.32, -136.242, 61.057, 156.046] to (-270.04, 305.9, -44.5) mm, rotated rx 180 ry 0 rz 0.01 deg; joints [37.321, -37.477, 89.187, -136.124, 61.042, 155.944]
  MoveC 5142 to (-269.47, 308.64, -44.5) mm, rotated rx 180 ry 0 rz 0.01 deg; joints [37.408, -37.418, 89.058, -136.007, 61.03, 155.844] to (-268.99, 311.39, -44.5) mm, rotated rx 180 ry 0 rz 0.01 deg; joints [37.494, -37.354, 88.919, -135.889, 61.013, 155.741]
  MoveC 5143 to (-269.73, 313.96, -44.5) mm, rotated rx 180 ry 0 rz 0.01 deg; joints [37.549, -37.247, 88.689, -135.785, 60.949, 155.615] to (-272.15, 315.07, -44.5) mm, rotated rx -180 ry 0 rz 0.01 deg; joints [37.529, -37.115, 88.41, -135.749, 60.835, 155.508]
  MoveL 5144 to (-375.8, 315.07, -44.5) mm, rotated rx 180 ry 0 rz 0.01 deg; joints [35.446, -32.6, 78.944, -135.809, 56.329, 152.615]
  MoveC 5145 to (-378.53, 313.94, -44.5) mm, rotated rx -180 ry 0 rz 0.01 deg; joints [35.363, -32.509, 78.755, -135.85, 56.219, 152.582] to (-379.65, 311.21, -44.5) mm, rotated rx 180 ry 0 rz 0.01 deg; joints [35.269, -32.544, 78.833, -135.97, 56.204, 152.675]
  MoveL 5146 to (-379.65, 88.69, -44.5) mm, rotated rx -180 ry 0 rz 0.01 deg; joints [28.83, -38.635, 91.984, -145.775, 59.058, 161.761]
  MoveC 5147 to (-378.57, 86.27, -44.5) mm, rotated rx -180 ry 0 rz 0.01 deg; joints [28.773, -38.736, 92.203, -145.877, 59.136, 161.871] to (-376.05, 85.43, -44.5) mm, rotated rx 180 ry 0 rz 0.01 deg; joints [28.789, -38.862, 92.473, -145.906, 59.261, 161.955]
  MoveC 5148 to (-355.38, 83.76, -44.5) mm, rotated rx 180 ry 0 rz 0.01 deg; joints [29.094, -39.771, 94.406, -145.908, 60.209, 162.448] to (-336.54, 75.06, -44.5) mm, rotated rx 180 ry 0 rz 0.01 deg; joints [29.151, -40.737, 96.48, -146.194, 61.146, 163.127]
  MoveC 5149 to (-332.72, 72.02, -44.5) mm, rotated rx 180 ry 0 rz 0.01 deg; joints [29.122, -40.958, 96.957, -146.303, 61.35, 163.305] to (-329.33, 68.51, -44.5) mm, rotated rx -180 ry 0 rz 0.01 deg; joints [29.07, -41.171, 97.418, -146.434, 61.541, 163.489]
  MoveC 5150 to (-326.23, 64.75, -44.5) mm, rotated rx 180 ry 0 rz 0.01 deg; joints [29.005, -41.376, 97.863, -146.577, 61.721, 163.674] to (-323.24, 60.9, -44.5) mm, rotated rx -180 ry 0 rz 0.01 deg; joints [28.935, -41.578, 98.302, -146.722, 61.898, 163.858]
  MoveL 5151 to (-303.16, 26.5, -44.5) mm, rotated rx 180 ry 0 rz 0.01 deg; joints [28.167, -43.074, 101.579, -148.049, 63.177, 165.33]
  MoveC 5152 to (-297.52, 12.02, -44.5) mm, rotated rx 180 ry 0 rz 0.01 deg; joints [27.785, -43.576, 102.69, -148.621, 63.591, 165.876] to (-296.45, -3.48, -44.5) mm, rotated rx 180 ry 0 rz 0.01 deg; joints [27.281, -43.914, 103.45, -149.271, 63.82, 166.365]
  MoveC 5153 to (-295.57, -6.04, -44.5) mm, rotated rx 180 ry 0 rz 0.01 deg; joints [27.209, -43.996, 103.633, -149.373, 63.888, 166.457] to (-293.08, -7.13, -44.5) mm, rotated rx 180 ry 0 rz 0.01 deg; joints [27.216, -44.112, 103.885, -149.4, 64.007, 166.531]
  MoveL 5154 to (-100.41, -7.13, -44.5) mm, rotated rx 180 ry 0 rz 0.01 deg; joints [31.014, -50.837, 118.711, -147.135, 71.778, 169.586]
  MoveC 5155 to (-97.91, -6.03, -44.5) mm, rotated rx -180 ry 0 rz 0.01 deg; joints [31.111, -50.896, 118.843, -147.049, 71.858, 169.595] to (-97.04, -3.45, -44.5) mm, rotated rx -180 ry 0 rz 0.01 deg; joints [31.225, -50.877, 118.793, -146.925, 71.856, 169.54]
  MoveC 5156 to (-97.12, 3.54, -44.5) mm, rotated rx 180 ry 0 rz 0.01 deg; joints [31.481, -50.747, 118.484, -146.63, 71.759, 169.352] to (-96.06, 10.45, -44.5) mm, rotated rx 180 ry 0 rz 0.01 deg; joints [31.757, -50.653, 118.257, -146.321, 71.706, 169.182]
  MoveC 5157 to (-94.17, 17.15, -44.5) mm, rotated rx -180 ry 0 rz 0.01 deg; joints [32.044, -50.588, 118.094, -146.008, 71.686, 169.029] to (-91.75, 23.69, -44.5) mm, rotated rx 180 ry 0 rz 0.01 deg; joints [32.336, -50.541, 117.975, -145.694, 71.689, 168.888]
  MoveL 5158 to (-72.01, 58.3, -44.5) mm, rotated rx 180 ry 0 rz 0.01 deg; joints [34.036, -50.486, 117.774, -143.922, 71.947, 168.237]
  MoveC 5159 to (-61.99, 70.84, -44.5) mm, rotated rx -180 ry 0 rz 0.01 deg; joints [34.72, -50.543, 117.875, -143.23, 72.139, 168.041] to (-48.71, 79.87, -44.5) mm, rotated rx -180 ry 0 rz 0.01 deg; joints [35.364, -50.764, 118.353, -142.622, 72.492, 167.997]
  MoveC 5160 to (-33.46, 84.78, -44.5) mm, rotated rx 180 ry 0 rz 0.01 deg; joints [35.919, -51.123, 119.151, -142.14, 72.968, 168.104] to (-17.45, 85.43, -44.5) mm, rotated rx 180 ry 0 rz 0.01 deg; joints [36.352, -51.586, 120.195, -141.808, 73.525, 168.347]
  MoveC 5161 to (-14.93, 86.26, -44.5) mm, rotated rx -180 ry 0 rz 0.01 deg; joints [36.446, -51.643, 120.322, -141.724, 73.601, 168.364] to (-13.86, 88.69, -44.5) mm, rotated rx -180 ry 0 rz 0.01 deg; joints [36.56, -51.624, 120.275, -141.604, 73.604, 168.311]
  MoveL 5162 to (-13.87, 311.22, -44.5) mm, rotated rx -180 ry 0 rz 0.01 deg; joints [43.616, -46.227, 107.9, -132.947, 70.494, 161.054]
  MoveC 5163 to (-14.99, 313.95, -44.5) mm, rotated rx 180 ry 0 rz 0.01 deg; joints [43.663, -46.118, 107.656, -132.865, 70.419, 160.935] to (-17.72, 315.08, -44.5) mm, rotated rx 180 ry 0 rz 0.01 deg; joints [43.622, -46.004, 107.408, -132.872, 70.313, 160.844]
  MoveL 5164 to (-121.36, 315.07, -44.5) mm, rotated rx -180 ry 0 rz 0.01 deg; joints [40.955, -42.694, 100.261, -134.445, 66.685, 158.866]
  MoveC 5165 to (-123.76, 313.97, -44.5) mm, rotated rx -180 ry 0 rz 0.01 deg; joints [40.865, -42.644, 100.156, -134.518, 66.612, 158.86] to (-124.5, 311.44, -44.5) mm, rotated rx 180 ry 0 rz 0.01 deg; joints [40.776, -42.691, 100.262, -134.626, 66.618, 158.942]
  MoveC 5166 to (-123.71, 306.39, -44.5) mm, rotated rx 180 ry 0 rz 0.01 deg; joints [40.653, -42.861, 100.634, -134.812, 66.714, 159.149] to (-122.84, 301.36, -44.5) mm, rotated rx 180 ry 0 rz 0.01 deg; joints [40.531, -43.033, 101.01, -134.997, 66.812, 159.356]
  MoveC 5167 to (-122.44, 296.24, -44.5) mm, rotated rx 180 ry 0 rz 0.01 deg; joints [40.394, -43.19, 101.354, -135.192, 66.894, 159.556] to (-123.1, 291.15, -44.5) mm, rotated rx 180 ry 0 rz 0.01 deg; joints [40.232, -43.309, 101.619, -135.399, 66.937, 159.733]
  MoveC 5168 to (-124.91, 284.21, -44.5) mm, rotated rx -180 ry 0 rz 0.01 deg; joints [39.988, -43.44, 101.912, -135.693, 66.963, 159.955] to (-127.02, 277.34, -44.5) mm, rotated rx 180 ry 0 rz 0.01 deg; joints [39.739, -43.557, 102.174, -135.989, 66.977, 160.167]
  MoveC 5169 to (-129.93, 270.75, -44.5) mm, rotated rx 180 ry 0 rz 0.01 deg; joints [39.476, -43.638, 102.359, -136.286, 66.957, 160.352] to (-134.04, 264.83, -44.5) mm, rotated rx 180 ry 0 rz 0.01 deg; joints [39.205, -43.658, 102.412, -136.571, 66.884, 160.488]
  MoveC 5170 to (-141.13, 257.49, -44.5) mm, rotated rx 180 ry 0 rz 0.01 deg; joints [38.82, -43.614, 102.328, -136.95, 66.718, 160.616] to (-149.11, 251.14, -44.5) mm, rotated rx -180 ry 0 rz 0.01 deg; joints [38.445, -43.509, 102.113, -137.301, 66.505, 160.691]
  MoveC 5171 to (-158.17, 246.34, -44.5) mm, rotated rx -180 ry 0 rz 0.01 deg; joints [38.091, -43.323, 101.72, -137.601, 66.228, 160.687] to (-168.11, 243.82, -44.5) mm, rotated rx -180 ry 0 rz 0.01 deg; joints [37.787, -43.043, 101.123, -137.817, 65.885, 160.583]
  MoveC 5172 to (-170.73, 243.47, -44.5) mm, rotated rx -180 ry 0 rz 0.01 deg; joints [37.716, -42.96, 100.946, -137.861, 65.79, 160.544] to (-173.34, 243.08, -44.5) mm, rotated rx 180 ry 0 rz 0.01 deg; joints [37.645, -42.878, 100.77, -137.906, 65.695, 160.506]
  MoveC 5173 to (-175.97, 242.79, -44.5) mm, rotated rx 180 ry 0 rz 0.01 deg; joints [37.576, -42.793, 100.588, -137.947, 65.599, 160.464] to (-178.62, 242.69, -44.5) mm, rotated rx -180 ry 0 rz 0.01 deg; joints [37.513, -42.702, 100.393, -137.98, 65.499, 160.415]
  MoveL 5174 to (-218.51, 242.92, -44.5) mm, rotated rx -180 ry 0 rz 0.01 deg; joints [36.632, -41.249, 97.284, -138.366, 63.944, 159.591]
  MoveC 5175 to (-228.86, 244.95, -44.5) mm, rotated rx -180 ry 0 rz 0.01 deg; joints [36.467, -40.808, 96.342, -138.372, 63.507, 159.296] to (-238.86, 248.28, -44.5) mm, rotated rx 180 ry 0 rz 0.01 deg; joints [36.349, -40.34, 95.34, -138.316, 63.063, 158.956]
  MoveC 5176 to (-248.13, 253.41, -44.5) mm, rotated rx -180 ry 0 rz 0.01 deg; joints [36.3, -39.845, 94.279, -138.173, 62.623, 158.556] to (-255.9, 260.62, -44.5) mm, rotated rx -180 ry 0 rz 0.01 deg; joints [36.343, -39.345, 93.206, -137.929, 62.214, 158.103]
  MoveC 5177 to (-262.3, 269.39, -44.5) mm, rotated rx 180 ry 0 rz 0.01 deg; joints [36.459, -38.848, 92.139, -137.605, 61.838, 157.612] to (-267.37, 279, -44.5) mm, rotated rx 180 ry 0 rz 0.01 deg; joints [36.625, -38.373, 91.12, -137.234, 61.505, 157.11]
  MoveC 5178 to (-270.4, 289.01, -44.5) mm, rotated rx 180 ry 0 rz 0.01 deg; joints [36.843, -37.962, 90.236, -136.832, 61.249, 156.632] to (-270.97, 299.46, -44.5) mm, rotated rx -180 ry 0 rz 0.01 deg; joints [37.122, -37.631, 89.522, -136.398, 61.089, 156.189]
  MoveC 5179 to (-269.46, 303.55, -44.5) mm, rotated rx 180 ry 0 rz 0.01 deg; joints [37.268, -37.57, 89.388, -136.22, 61.097, 156.056] to (-265.97, 306.15, -44.5) mm, rotated rx -180 ry 0 rz 0.01 deg; joints [37.413, -37.633, 89.515, -136.094, 61.207, 156.034]
  MoveC 5180 to (-262.4, 308.53, -44.5) mm, rotated rx 180 ry 0 rz 0.01 deg; joints [37.555, -37.705, 89.663, -135.978, 61.322, 156.022] to (-260.27, 312.25, -44.5) mm, rotated rx -180 ry 0 rz 0.01 deg; joints [37.703, -37.678, 89.601, -135.811, 61.36, 155.92]
  MoveC 5181 to (-258.79, 316.42, -44.5) mm, rotated rx 180 ry 0 rz 0.01 deg; joints [37.85, -37.611, 89.454, -135.63, 61.366, 155.782] to (-256.86, 320.4, -44.5) mm, rotated rx -180 ry 0 rz 0.01 deg; joints [38, -37.567, 89.356, -135.455, 61.392, 155.663]
  MoveC 5182 to (-256.89, 322.65, -44.5) mm, rotated rx 180 ry 0 rz 0.01 deg; joints [38.061, -37.497, 89.205, -135.361, 61.362, 155.568] to (-258.85, 323.77, -44.5) mm, rotated rx 180 ry 0 rz 0.01 deg; joints [38.05, -37.385, 88.967, -135.324, 61.267, 155.473]
  MoveL 5183 to (-384.5, 323.76, -44.5) mm, rotated rx -180 ry 0 rz 0.01 deg; joints [35.513, -31.9, 77.472, -135.375, 55.81, 151.924]
  MoveC 5184 to (-387.22, 322.63, -44.5) mm, rotated rx -180 ry 0 rz 0.01 deg; joints [35.431, -31.807, 77.28, -135.414, 55.699, 151.889] to (-388.35, 319.91, -44.5) mm, rotated rx 180 ry 0 rz 0.01 deg; joints [35.337, -31.844, 77.36, -135.534, 55.684, 151.983]
  MoveL 5185 to (-388.34, 76.97, -44.5) mm, rotated rx -180 ry 0 rz 0.01 deg; joints [28.319, -38.525, 91.772, -146.302, 58.803, 161.99]
  MoveC 5186 to (-387.22, 74.74, -44.5) mm, rotated rx 180 ry 0 rz 0.01 deg; joints [28.268, -38.623, 91.985, -146.397, 58.881, 162.093] to (-384.76, 74.3, -44.5) mm, rotated rx 180 ry 0 rz 0.01 deg; joints [28.296, -38.739, 92.231, -146.41, 58.999, 162.162]
  MoveC 5187 to (-382.03, 75.17, -44.5) mm, rotated rx 180 ry 0 rz 0.01 deg; joints [28.369, -38.837, 92.437, -146.365, 59.113, 162.189] to (-379.33, 76.14, -44.5) mm, rotated rx 180 ry 0 rz 0.01 deg; joints [28.444, -38.931, 92.634, -146.316, 59.224, 162.213]
  MoveC 5188 to (-376.56, 76.92, -44.5) mm, rotated rx 180 ry 0 rz 0.01 deg; joints [28.516, -39.032, 92.846, -146.274, 59.34, 162.244] to (-373.7, 77.21, -44.5) mm, rotated rx -180 ry 0 rz 0.01 deg; joints [28.574, -39.147, 93.091, -146.253, 59.466, 162.294]
  MoveC 5189 to (-364.55, 76.72, -44.5) mm, rotated rx 180 ry 0 rz 0.01 deg; joints [28.715, -39.544, 93.935, -146.244, 59.884, 162.502] to (-355.54, 75.02, -44.5) mm, rotated rx -180 ry 0 rz 0.01 deg; joints [28.817, -39.957, 94.818, -146.282, 60.307, 162.746]
  MoveC 5190 to (-346.97, 71.64, -44.5) mm, rotated rx 180 ry 0 rz 0.01 deg; joints [28.859, -40.385, 95.735, -146.39, 60.728, 163.035] to (-339.47, 66.3, -44.5) mm, rotated rx -180 ry 0 rz 0.01 deg; joints [28.821, -40.808, 96.646, -146.582, 61.123, 163.364]
  MoveC 5191 to (-336.49, 63.42, -44.5) mm, rotated rx -180 ry 0 rz 0.01 deg; joints [28.781, -40.991, 97.042, -146.689, 61.289, 163.519] to (-333.67, 60.38, -44.5) mm, rotated rx -180 ry 0 rz 0.01 deg; joints [28.733, -41.17, 97.43, -146.803, 61.449, 163.675]
  MoveC 5192 to (-331.09, 57.13, -44.5) mm, rotated rx 180 ry 0 rz 0.01 deg; joints [28.674, -41.343, 97.806, -146.927, 61.601, 163.832] to (-328.84, 53.64, -44.5) mm, rotated rx 180 ry 0 rz 0.01 deg; joints [28.601, -41.506, 98.163, -147.063, 61.741, 163.99]
  MoveL 5193 to (-309.59, 19.91, -44.5) mm, rotated rx -180 ry 0 rz 0.01 deg; joints [27.835, -42.954, 101.334, -148.374, 62.978, 165.422]
  MoveC 5194 to (-307.47, 14.26, -44.5) mm, rotated rx 180 ry 0 rz 0.01 deg; joints [27.684, -43.148, 101.761, -148.599, 63.137, 165.634] to (-305.74, 8.48, -44.5) mm, rotated rx -180 ry 0 rz 0.01 deg; joints [27.521, -43.327, 102.159, -148.832, 63.279, 165.842]
  MoveC 5195 to (-304.76, 2.51, -44.5) mm, rotated rx 180 ry 0 rz 0.01 deg; joints [27.338, -43.479, 102.5, -149.078, 63.392, 166.042] to (-304.91, -3.54, -44.5) mm, rotated rx -180 ry 0 rz 0.01 deg; joints [27.132, -43.589, 102.747, -149.336, 63.456, 166.223]
  MoveC 5196 to (-305.2, -5.77, -44.5) mm, rotated rx -180 ry 0 rz 0.01 deg; joints [27.052, -43.62, 102.818, -149.433, 63.47, 166.285] to (-305.52, -7.98, -44.5) mm, rotated rx 180 ry 0 rz 0.01 deg; joints [26.971, -43.649, 102.886, -149.529, 63.482, 166.347]
  MoveC 5197 to (-305.89, -10.19, -44.5) mm, rotated rx 180 ry 0 rz 0.01 deg; joints [26.89, -43.675, 102.948, -149.626, 63.492, 166.407] to (-306.35, -12.38, -44.5) mm, rotated rx 180 ry 0 rz 0.01 deg; joints [26.808, -43.699, 103.002, -149.723, 63.498, 166.465]
  MoveC 5198 to (-305.81, -14.77, -44.5) mm, rotated rx 180 ry 0 rz 0.01 deg; joints [26.736, -43.764, 103.148, -149.82, 63.549, 166.545] to (-303.61, -15.83, -44.5) mm, rotated rx 180 ry 0 rz 0.01 deg; joints [26.738, -43.869, 103.377, -149.849, 63.656, 166.614]
  MoveL 5199 to (-89.9, -15.83, -44.5) mm, rotated rx -180 ry 0 rz 0.01 deg; joints [30.926, -51.325, 119.835, -147.338, 72.294, 169.976]
  MoveC 5200 to (-87.7, -14.77, -44.5) mm, rotated rx 180 ry 0 rz 0.01 deg; joints [31.015, -51.375, 119.946, -147.257, 72.363, 169.982] to (-87.16, -12.38, -44.5) mm, rotated rx -180 ry 0 rz 0.01 deg; joints [31.116, -51.35, 119.883, -147.146, 72.351, 169.928]
  MoveC 5201 to (-88.16, -6.74, -44.5) mm, rotated rx 180 ry 0 rz 0.01 deg; joints [31.303, -51.217, 119.569, -146.922, 72.237, 169.764] to (-88.59, -1.03, -44.5) mm, rotated rx -180 ry 0 rz 0.01 deg; joints [31.505, -51.1, 119.291, -146.687, 72.143, 169.606]
  MoveC 5202 to (-88.4, 4.69, -44.5) mm, rotated rx -180 ry 0 rz 0.01 deg; joints [31.72, -51.001, 119.055, -146.441, 72.073, 169.456] to (-87.54, 10.36, -44.5) mm, rotated rx -180 ry 0 rz 0.01 deg; joints [31.947, -50.924, 118.867, -146.187, 72.028, 169.317]
  MoveC 5203 to (-86.7, 13.55, -44.5) mm, rotated rx 180 ry 0 rz 0.01 deg; joints [32.083, -50.891, 118.786, -146.039, 72.016, 169.244] to (-85.56, 16.64, -44.5) mm, rotated rx -180 ry 0 rz 0.01 deg; joints [32.222, -50.869, 118.728, -145.89, 72.016, 169.178]
  MoveC 5204 to (-84.19, 19.64, -44.5) mm, rotated rx -180 ry 0 rz 0.01 deg; joints [32.363, -50.856, 118.692, -145.741, 72.027, 169.118] to (-82.63, 22.55, -44.5) mm, rotated rx 180 ry 0 rz 0.01 deg; joints [32.504, -50.85, 118.672, -145.593, 72.045, 169.063]
  MoveL 5205 to (-63.06, 56.07, -44.5) mm, rotated rx 180 ry 0 rz 0.01 deg; joints [34.172, -50.807, 118.501, -143.859, 72.305, 168.444]
  MoveC 5206 to (-53.48, 66.04, -44.5) mm, rotated rx 180 ry 0 rz 0.01 deg; joints [34.759, -50.901, 118.691, -143.277, 72.515, 168.316] to (-41.96, 73.7, -44.5) mm, rotated rx 180 ry 0 rz 0.01 deg; joints [35.315, -51.095, 119.112, -142.753, 72.822, 168.284]
  MoveC 5207 to (-28.52, 77.64, -44.5) mm, rotated rx 180 ry 0 rz 0.01 deg; joints [35.793, -51.418, 119.833, -142.34, 73.245, 168.39] to (-14.58, 76.24, -44.5) mm, rotated rx -180 ry 0 rz 0.01 deg; joints [36.101, -51.859, 120.836, -142.129, 73.758, 168.657]
  MoveC 5208 to (-13.11, 75.77, -44.5) mm, rotated rx 180 ry 0 rz 0.01 deg; joints [36.123, -51.912, 120.956, -142.119, 73.816, 168.694] to (-11.66, 75.26, -44.5) mm, rotated rx -180 ry 0 rz 0.01 deg; joints [36.142, -51.965, 121.078, -142.111, 73.875, 168.732]
  MoveC 5209 to (-10.21, 74.74, -44.5) mm, rotated rx 180 ry 0 rz 0.01 deg; joints [36.161, -52.018, 121.2, -142.104, 73.933, 168.77] to (-8.75, 74.27, -44.5) mm, rotated rx -180 ry 0 rz 0.01 deg; joints [36.183, -52.07, 121.32, -142.094, 73.991, 168.807]
  MoveC 5210 to (-6.29, 74.7, -44.5) mm, rotated rx -180 ry 0 rz 0.01 deg; joints [36.262, -52.133, 121.462, -142.027, 74.071, 168.835] to (-5.16, 76.93, -44.5) mm, rotated rx 180 ry 0 rz 0.01 deg; joints [36.371, -52.12, 121.428, -141.913, 74.078, 168.79]
  MoveL 5211 to (-5.17, 319.92, -44.5) mm, rotated rx 180 ry 0 rz 0.01 deg; joints [44.101, -46.244, 107.923, -132.467, 70.667, 160.894]
  MoveC 5212 to (-6.3, 322.64, -44.5) mm, rotated rx 180 ry 0 rz 0.01 deg; joints [44.147, -46.134, 107.678, -132.387, 70.593, 160.774] to (-9.02, 323.77, -44.5) mm, rotated rx 180 ry 0 rz 0.01 deg; joints [44.104, -46.021, 107.43, -132.394, 70.487, 160.683]
  MoveL 5213 to (-134.6, 323.77, -44.5) mm, rotated rx -180 ry 0 rz 0.01 deg; joints [40.877, -41.991, 98.744, -134.269, 66.085, 158.263]
  MoveC 5214 to (-136.59, 322.65, -44.5) mm, rotated rx -180 ry 0 rz 0.01 deg; joints [40.798, -41.955, 98.669, -134.336, 66.027, 158.265] to (-136.66, 320.37, -44.5) mm, rotated rx -180 ry 0 rz 0.01 deg; joints [40.733, -42.019, 98.808, -134.426, 66.054, 158.352]
  MoveC 5215 to (-133.78, 313.94, -44.5) mm, rotated rx 180 ry 0 rz 0.01 deg; joints [40.622, -42.303, 99.426, -134.643, 66.245, 158.658] to (-131.67, 307.22, -44.5) mm, rotated rx -180 ry 0 rz 0.01 deg; joints [40.483, -42.567, 100.002, -134.879, 66.411, 158.958]
  MoveC 5216 to (-130.77, 300.2, -44.5) mm, rotated rx -180 ry 0 rz 0.01 deg; joints [40.305, -42.797, 100.504, -135.143, 66.537, 159.242] to (-131.56, 293.16, -44.5) mm, rotated rx 180 ry 0 rz 0.01 deg; joints [40.085, -42.967, 100.88, -135.428, 66.601, 159.491]
  MoveC 5217 to (-133.88, 284.87, -44.5) mm, rotated rx 180 ry 0 rz 0.01 deg; joints [39.791, -43.118, 101.218, -135.782, 66.625, 159.754] to (-136.87, 276.79, -44.5) mm, rotated rx -180 ry 0 rz 0.01 deg; joints [39.486, -43.238, 101.488, -136.136, 66.621, 159.994]
  MoveC 5218 to (-141.24, 269.3, -44.5) mm, rotated rx -180 ry 0 rz 0.01 deg; joints [39.164, -43.292, 101.617, -136.486, 66.558, 160.184] to (-147.44, 263.23, -44.5) mm, rotated rx 180 ry 0 rz 0.01 deg; joints [38.84, -43.243, 101.522, -136.802, 66.407, 160.284]
  MoveC 5219 to (-154.51, 258.58, -44.5) mm, rotated rx -180 ry 0 rz 0.01 deg; joints [38.537, -43.124, 101.274, -137.071, 66.204, 160.315] to (-162.07, 254.79, -44.5) mm, rotated rx 180 ry 0 rz 0.01 deg; joints [38.25, -42.962, 100.933, -137.311, 65.969, 160.303]
  MoveC 5220 to (-170.17, 252.24, -44.5) mm, rotated rx -180 ry 0 rz 0.01 deg; joints [37.988, -42.746, 100.473, -137.504, 65.696, 160.235] to (-178.62, 251.38, -44.5) mm, rotated rx 180 ry 0 rz 0.01 deg; joints [37.769, -42.471, 99.883, -137.632, 65.385, 160.097]
  MoveL 5221 to (-217.39, 251.55, -44.5) mm, rotated rx -180 ry 0 rz 0.01 deg; joints [36.908, -41.058, 96.863, -138.005, 63.876, 159.292]
  MoveC 5222 to (-226.18, 253.22, -44.5) mm, rotated rx -180 ry 0 rz 0.01 deg; joints [36.766, -40.685, 96.065, -138.012, 63.506, 159.041] to (-234.7, 255.91, -44.5) mm, rotated rx -180 ry 0 rz 0.01 deg; joints [36.659, -40.29, 95.22, -137.971, 63.131, 158.755]
  MoveC 5223 to (-242.64, 260.15, -44.5) mm, rotated rx 180 ry 0 rz 0.01 deg; joints [36.611, -39.87, 94.322, -137.856, 62.757, 158.418] to (-249.27, 266.24, -44.5) mm, rotated rx -180 ry 0 rz 0.01 deg; joints [36.645, -39.445, 93.411, -137.653, 62.41, 158.033]
  MoveC 5224 to (-252.98, 271.05, -44.5) mm, rotated rx -180 ry 0 rz 0.01 deg; joints [36.703, -39.166, 92.811, -137.479, 62.197, 157.76] to (-256.24, 276.18, -44.5) mm, rotated rx -180 ry 0 rz 0.01 deg; joints [36.78, -38.893, 92.225, -137.287, 61.997, 157.482]
  MoveC 5225 to (-258.87, 281.67, -44.5) mm, rotated rx 180 ry 0 rz 0.01 deg; joints [36.879, -38.633, 91.665, -137.075, 61.818, 157.202] to (-260.64, 287.5, -44.5) mm, rotated rx 180 ry 0 rz 0.01 deg; joints [37.006, -38.395, 91.152, -136.843, 61.67, 156.926]
  MoveC 5226 to (-261.84, 295.85, -44.5) mm, rotated rx 180 ry 0 rz 0.01 deg; joints [37.215, -38.103, 90.523, -136.503, 61.511, 156.558] to (-261.76, 304.29, -44.5) mm, rotated rx -180 ry 0 rz 0.01 deg; joints [37.451, -37.856, 89.99, -136.151, 61.404, 156.213]
  MoveC 5227 to (-261.22, 308.31, -44.5) mm, rotated rx -180 ry 0 rz 0.01 deg; joints [37.574, -37.758, 89.777, -135.98, 61.373, 156.06] to (-260.27, 312.25, -44.5) mm, rotated rx -180 ry 0 rz 0.01 deg; joints [37.703, -37.678, 89.601, -135.811, 61.36, 155.92]
  MoveC 5228 to (-258.08, 315.41, -44.5) mm, rotated rx -180 ry 0 rz 0.01 deg; joints [37.837, -37.67, 89.579, -135.669, 61.408, 155.841] to (-254.44, 316.65, -44.5) mm, rotated rx 180 ry 0 rz 0.01 deg; joints [37.949, -37.777, 89.804, -135.598, 61.541, 155.878]
  MoveC 5229 to (-250.79, 317.66, -44.5) mm, rotated rx 180 ry 0 rz 0.01 deg; joints [38.056, -37.891, 90.043, -135.536, 61.675, 155.925] to (-248.13, 320.34, -44.5) mm, rotated rx -180 ry 0 rz 0.01 deg; joints [38.187, -37.915, 90.089, -135.41, 61.748, 155.878]
  MoveC 5230 to (-247.43, 321.55, -44.5) mm, rotated rx -180 ry 0 rz 0.01 deg; joints [38.235, -37.906, 90.069, -135.357, 61.76, 155.845] to (-246.73, 322.74, -44.5) mm, rotated rx 180 ry 0 rz 0.01 deg; joints [38.283, -37.897, 90.048, -135.303, 61.773, 155.812]
  MoveC 5231 to (-244.61, 325.94, -44.5) mm, rotated rx -180 ry 0 rz 0.01 deg; joints [38.417, -37.883, 90.015, -135.159, 61.817, 155.73] to (-242.15, 328.88, -44.5) mm, rotated rx -180 ry 0 rz 0.01 deg; joints [38.551, -37.89, 90.026, -135.023, 61.877, 155.667]
  MoveC 5232 to (-241.81, 330.8, -44.5) mm, rotated rx 180 ry 0 rz 0.01 deg; joints [38.611, -37.845, 89.927, -134.942, 61.866, 155.594] to (-243.44, 331.87, -44.5) mm, rotated rx 180 ry 0 rz 0.01 deg; joints [38.604, -37.748, 89.721, -134.907, 61.786, 155.51]
  MoveL 5233 to (-392.6, 331.87, -44.5) mm, rotated rx -180 ry 0 rz 0.01 deg; joints [35.574, -31.234, 76.074, -134.957, 55.321, 151.261]
  MoveC 5234 to (-395.33, 330.74, -44.5) mm, rotated rx -180 ry 0 rz 0.01 deg; joints [35.493, -31.14, 75.878, -134.993, 55.209, 151.223] to (-396.45, 328.01, -44.5) mm, rotated rx -180 ry 0 rz 0.01 deg; joints [35.399, -31.177, 75.961, -135.113, 55.194, 151.319]
  MoveL 5235 to (-396.45, 62.47, -44.5) mm, rotated rx -180 ry 0 rz 0.01 deg; joints [27.732, -38.496, 91.735, -146.948, 58.603, 162.328]
  MoveC 5236 to (-395.33, 60.7, -44.5) mm, rotated rx 180 ry 0 rz 0.01 deg; joints [27.695, -38.583, 91.923, -147.023, 58.676, 162.414] to (-393.25, 60.93, -44.5) mm, rotated rx -180 ry 0 rz 0.01 deg; joints [27.736, -38.668, 92.103, -147.008, 58.769, 162.451]
  MoveC 5237 to (-391.49, 62.33, -44.5) mm, rotated rx -180 ry 0 rz 0.01 deg; joints [27.809, -38.713, 92.197, -146.944, 58.833, 162.439] to (-389.74, 63.74, -44.5) mm, rotated rx 180 ry 0 rz 0.01 deg; joints [27.882, -38.758, 92.289, -146.879, 58.897, 162.427]
  MoveC 5238 to (-387.86, 64.98, -44.5) mm, rotated rx -180 ry 0 rz 0.01 deg; joints [27.953, -38.812, 92.401, -146.82, 58.968, 162.423] to (-385.77, 65.84, -44.5) mm, rotated rx -180 ry 0 rz 0.01 deg; joints [28.014, -38.883, 92.551, -146.778, 59.054, 162.438]
  MoveL 5239 to (-376.06, 68.68, -44.5) mm, rotated rx 180 ry 0 rz 0.01 deg; joints [28.266, -39.235, 93.293, -146.628, 59.462, 162.542]
  MoveC 5240 to (-371.03, 69.52, -44.5) mm, rotated rx 180 ry 0 rz 0.01 deg; joints [28.378, -39.429, 93.705, -146.576, 59.679, 162.618] to (-365.95, 69.18, -44.5) mm, rotated rx 180 ry 0 rz 0.01 deg; joints [28.454, -39.651, 94.176, -146.573, 59.912, 162.734]
  MoveC 5241 to (-358.95, 67.5, -44.5) mm, rotated rx 180 ry 0 rz 0.01 deg; joints [28.521, -39.98, 94.879, -146.618, 60.246, 162.935] to (-352.17, 65.09, -44.5) mm, rotated rx -180 ry 0 rz 0.01 deg; joints [28.561, -40.313, 95.594, -146.693, 60.576, 163.153]
  MoveC 5242 to (-345.91, 61.44, -44.5) mm, rotated rx 180 ry 0 rz 0.01 deg; joints [28.553, -40.649, 96.317, -146.82, 60.898, 163.401] to (-340.81, 56.29, -44.5) mm, rotated rx 180 ry 0 rz 0.01 deg; joints [28.477, -40.967, 97.004, -147.015, 61.184, 163.673]
  MoveC 5243 to (-339.54, 54.64, -44.5) mm, rotated rx 180 ry 0 rz 0.01 deg; joints [28.446, -41.054, 97.192, -147.079, 61.26, 163.752] to (-338.23, 53.02, -44.5) mm, rotated rx 180 ry 0 rz 0.01 deg; joints [28.417, -41.141, 97.382, -147.141, 61.337, 163.831]
  MoveC 5244 to (-336.97, 51.36, -44.5) mm, rotated rx 180 ry 0 rz 0.01 deg; joints [28.385, -41.226, 97.568, -147.205, 61.412, 163.91] to (-335.86, 49.6, -44.5) mm, rotated rx -180 ry 0 rz 0.01 deg; joints [28.348, -41.308, 97.746, -147.274, 61.482, 163.989]
  MoveL 5245 to (-317.07, 16.81, -44.5) mm, rotated rx 180 ry 0 rz 0.01 deg; joints [27.602, -42.722, 100.839, -148.556, 62.691, 165.385]
  MoveC 5246 to (-314.65, 9.86, -44.5) mm, rotated rx -180 ry 0 rz 0.01 deg; joints [27.413, -42.953, 101.35, -148.835, 62.878, 165.644] to (-313.02, 2.69, -44.5) mm, rotated rx 180 ry 0 rz 0.01 deg; joints [27.201, -43.155, 101.799, -149.128, 63.033, 165.893]
  MoveC 5247 to (-312.74, -4.71, -44.5) mm, rotated rx -180 ry 0 rz 0.01 deg; joints [26.958, -43.306, 102.14, -149.441, 63.132, 166.124] to (-314.34, -11.93, -44.5) mm, rotated rx 180 ry 0 rz 0.01 deg; joints [26.687, -43.379, 102.312, -149.76, 63.146, 166.315]
  MoveC 5248 to (-315.2, -14.16, -44.5) mm, rotated rx -180 ry 0 rz 0.01 deg; joints [26.597, -43.387, 102.334, -149.86, 63.134, 166.368] to (-316.14, -16.36, -44.5) mm, rotated rx 180 ry 0 rz 0.01 deg; joints [26.507, -43.392, 102.347, -149.96, 63.119, 166.418]
  MoveC 5249 to (-317.18, -18.51, -44.5) mm, rotated rx 180 ry 0 rz 0.01 deg; joints [26.416, -43.391, 102.35, -150.059, 63.099, 166.465] to (-318.34, -20.6, -44.5) mm, rotated rx 180 ry 0 rz 0.01 deg; joints [26.326, -43.384, 102.339, -150.156, 63.072, 166.509]
  MoveC 5250 to (-318.36, -22.82, -44.5) mm, rotated rx -180 ry 0 rz 0.01 deg; joints [26.25, -43.424, 102.43, -150.251, 63.097, 166.575] to (-316.44, -23.93, -44.5) mm, rotated rx -180 ry 0 rz 0.01 deg; joints [26.245, -43.519, 102.638, -150.285, 63.193, 166.64]
  MoveL 5251 to (-77.11, -23.93, -44.5) mm, rotated rx 180 ry 0 rz 0.01 deg; joints [30.909, -51.868, 121.087, -147.475, 72.889, 170.382]
  MoveC 5252 to (-75.17, -22.82, -44.5) mm, rotated rx -180 ry 0 rz 0.01 deg; joints [30.995, -51.908, 121.177, -147.395, 72.947, 170.383] to (-75.17, -20.58, -44.5) mm, rotated rx -180 ry 0 rz 0.01 deg; joints [31.079, -51.869, 121.082, -147.299, 72.916, 170.325]
  MoveC 5253 to (-77.64, -15.75, -44.5) mm, rotated rx 180 ry 0 rz 0.01 deg; joints [31.205, -51.707, 120.702, -147.133, 72.757, 170.162] to (-79.6, -10.7, -44.5) mm, rotated rx 180 ry 0 rz 0.01 deg; joints [31.35, -51.556, 120.347, -146.95, 72.614, 170]
  MoveC 5254 to (-80.78, -5.38, -44.5) mm, rotated rx -180 ry 0 rz 0.01 deg; joints [31.521, -51.424, 120.034, -146.743, 72.497, 169.842] to (-80.86, 0.06, -44.5) mm, rotated rx -180 ry 0 rz 0.01 deg; joints [31.721, -51.322, 119.792, -146.513, 72.419, 169.697]
  MoveC 5255 to (-80.24, 4.84, -44.5) mm, rotated rx 180 ry 0 rz 0.01 deg; joints [31.912, -51.254, 119.626, -146.3, 72.377, 169.579] to (-79.24, 9.56, -44.5) mm, rotated rx 180 ry 0 rz 0.01 deg; joints [32.108, -51.198, 119.489, -146.084, 72.35, 169.468]
  MoveC 5256 to (-77.73, 14.15, -44.5) mm, rotated rx 180 ry 0 rz 0.01 deg; joints [32.312, -51.16, 119.392, -145.865, 72.343, 169.368] to (-75.61, 18.49, -44.5) mm, rotated rx 180 ry 0 rz 0.01 deg; joints [32.52, -51.145, 119.348, -145.646, 72.363, 169.284]
  MoveL 5257 to (-56.64, 51.13, -44.5) mm, rotated rx -180 ry 0 rz 0.01 deg; joints [34.151, -51.102, 119.177, -143.952, 72.609, 168.686]
  MoveC 5258 to (-51.79, 56.78, -44.5) mm, rotated rx -180 ry 0 rz 0.01 deg; joints [34.471, -51.138, 119.246, -143.631, 72.706, 168.606] to (-46.38, 61.89, -44.5) mm, rotated rx 180 ry 0 rz 0.01 deg; joints [34.787, -51.2, 119.375, -143.321, 72.829, 168.549]
  MoveC 5259 to (-40.08, 65.95, -44.5) mm, rotated rx -180 ry 0 rz 0.01 deg; joints [35.088, -51.309, 119.612, -143.038, 72.999, 168.536] to (-32.94, 68.22, -44.5) mm, rotated rx -180 ry 0 rz 0.01 deg; joints [35.348, -51.478, 119.988, -142.811, 73.222, 168.587]
  MoveC 5260 to (-25.14, 69.09, -44.5) mm, rotated rx 180 ry 0 rz 0.01 deg; joints [35.576, -51.693, 120.473, -142.627, 73.487, 168.688] to (-17.3, 68.93, -44.5) mm, rotated rx -180 ry 0 rz 0.01 deg; joints [35.771, -51.928, 121.008, -142.483, 73.767, 168.82]
  MoveC 5261 to (-9.6, 67.09, -44.5) mm, rotated rx -180 ry 0 rz 0.01 deg; joints [35.904, -52.191, 121.61, -142.407, 74.065, 168.996] to (-2.77, 63.09, -44.5) mm, rotated rx 180 ry 0 rz 0.01 deg; joints [35.938, -52.47, 122.256, -142.436, 74.363, 169.219]
  MoveC 5262 to (-2.13, 62.56, -44.5) mm, rotated rx -180 ry 0 rz 0.01 deg; joints [35.936, -52.499, 122.324, -142.445, 74.394, 169.244] to (-1.51, 62, -44.5) mm, rotated rx -180 ry 0 rz 0.01 deg; joints [35.932, -52.528, 122.392, -142.455, 74.424, 169.27]
  MoveC 5263 to (-0.89, 61.45, -44.5) mm, rotated rx 180 ry 0 rz 0.01 deg; joints [35.928, -52.557, 122.46, -142.465, 74.453, 169.295] to (-0.24, 60.92, -44.5) mm, rotated rx -180 ry 0 rz 0.01 deg; joints [35.926, -52.586, 122.528, -142.474, 74.484, 169.321]
  MoveC 5264 to (1.83, 60.68, -44.5) mm, rotated rx 180 ry 0 rz 0.01 deg; joints [35.972, -52.651, 122.676, -142.442, 74.56, 169.361] to (2.94, 62.44, -44.5) mm, rotated rx -180 ry 0 rz 0.01 deg; joints [36.065, -52.648, 122.665, -142.347, 74.573, 169.33]
  MoveL 5265 to (2.93, 328.02, -44.5) mm, rotated rx 180 ry 0 rz 0.01 deg; joints [44.552, -46.256, 107.935, -132.02, 70.826, 160.742]
  MoveC 5266 to (1.8, 330.75, -44.5) mm, rotated rx 180 ry 0 rz 0.01 deg; joints [44.597, -46.145, 107.69, -131.94, 70.752, 160.621] to (-0.92, 331.88, -44.5) mm, rotated rx -180 ry 0 rz 0.01 deg; joints [44.554, -46.032, 107.443, -131.948, 70.647, 160.53]
  MoveL 5267 to (-150.07, 331.87, -44.5) mm, rotated rx -180 ry 0 rz 0.01 deg; joints [40.731, -41.216, 97.077, -134.127, 65.405, 157.624]
  MoveC 5268 to (-151.7, 330.8, -44.5) mm, rotated rx 180 ry 0 rz 0.01 deg; joints [40.663, -41.191, 97.024, -134.187, 65.359, 157.631] to (-151.37, 328.88, -44.5) mm, rotated rx -180 ry 0 rz 0.01 deg; joints [40.618, -41.259, 97.172, -134.259, 65.396, 157.714]
  MoveC 5269 to (-146.02, 321.99, -44.5) mm, rotated rx 180 ry 0 rz 0.01 deg; joints [40.553, -41.648, 98.012, -134.471, 65.686, 158.096] to (-142.04, 314.22, -44.5) mm, rotated rx 180 ry 0 rz 0.01 deg; joints [40.431, -42.01, 98.799, -134.73, 65.936, 158.479]
  MoveC 5270 to (-139.69, 305.81, -44.5) mm, rotated rx 180 ry 0 rz 0.01 deg; joints [40.25, -42.332, 99.501, -135.032, 66.134, 158.849] to (-139.16, 297.09, -44.5) mm, rotated rx 180 ry 0 rz 0.01 deg; joints [40.015, -42.597, 100.081, -135.367, 66.268, 159.191]
  MoveC 5271 to (-141.74, 285.04, -44.5) mm, rotated rx -180 ry 0 rz 0.01 deg; joints [39.608, -42.844, 100.63, -135.872, 66.332, 159.591] to (-148.06, 274.47, -44.5) mm, rotated rx -180 ry 0 rz 0.01 deg; joints [39.153, -42.917, 100.803, -136.365, 66.236, 159.858]
  MoveC 5272 to (-157.21, 266.29, -44.5) mm, rotated rx 180 ry 0 rz 0.01 deg; joints [38.7, -42.822, 100.613, -136.797, 66.001, 159.978] to (-168.25, 260.93, -44.5) mm, rotated rx -180 ry 0 rz 0.01 deg; joints [38.287, -42.581, 100.104, -137.136, 65.655, 159.954]
